Yaskawa INFORM job: s1234_1.JBI

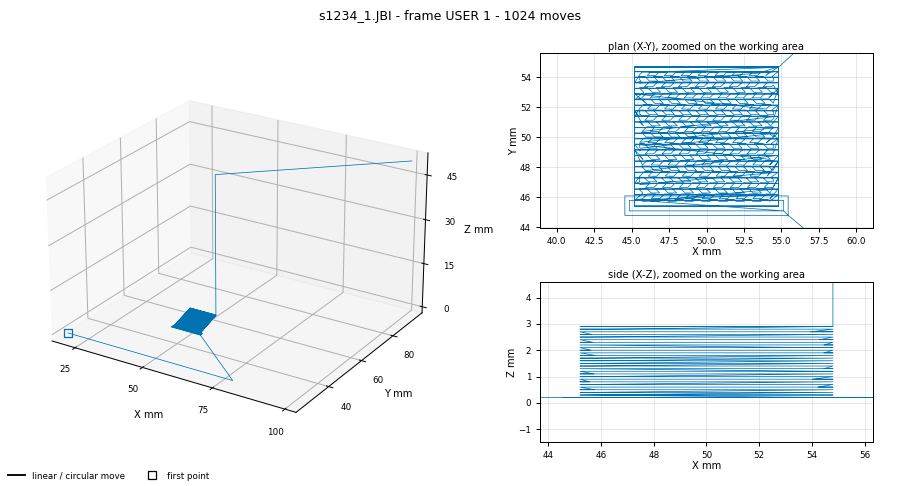
[picture p0: tool path of s1234_1.JBI in frame USER 1, 1024 of 1024 moves have a stored position in this frame; points joined in program order, loops and branches not executed]
/JOB
//NAME s1234_1
//POS
///NPOS 1024,0,0,0,0,0
///USER 1
///TOOL 1
///POSTYPE USER
///RECTAN
///RCONF 1,0,0,0,0,0
C00000=20.000,24.400,0.200,0.000,-180.000,-30.000
C00001=80.000,24.400,0.200,0.000,-180.000,-30.000
C00002=80.000,24.400,0.200,0.000,-180.000,-30.000
C00003=55.450,44.784,0.200,0.000,-180.000,-30.000
C00004=55.450,44.784,0.200,0.000,-180.000,-30.000
C00005=55.450,46.080,0.200,0.000,-180.000,-30.000
C00006=44.550,46.080,0.200,0.000,-180.000,-30.000
C00007=44.550,44.784,0.200,0.000,-180.000,-30.000
C00008=55.450,44.784,0.200,0.000,-180.000,-30.000
C00009=55.150,45.084,0.200,0.000,-180.000,-30.000
C00010=55.150,45.780,0.200,0.000,-180.000,-30.000
C00011=44.850,45.780,0.200,0.000,-180.000,-30.000
C00012=44.850,45.084,0.200,0.000,-180.000,-30.000
C00013=55.150,45.084,0.200,0.000,-180.000,-30.000
C00014=55.150,45.084,0.200,0.000,-180.000,-30.000
C00015=45.200,45.803,0.300,0.000,-180.000,-30.000
C00016=45.200,45.803,0.300,0.000,-180.000,-30.000
C00017=45.200,45.407,0.300,0.000,-180.000,-30.000
C00018=54.800,45.407,0.300,0.000,-180.000,-30.000
C00019=54.800,45.803,0.300,0.000,-180.000,-30.000
C00020=45.200,45.803,0.300,0.000,-180.000,-30.000
C00021=45.200,45.803,0.300,0.000,-180.000,-30.000
C00022=54.800,46.176,0.400,0.000,-180.000,-30.000
C00023=54.800,46.176,0.400,0.000,-180.000,-30.000
C00024=45.200,46.176,0.400,0.000,-180.000,-30.000
C00025=45.200,45.380,0.400,0.000,-180.000,-30.000
C00026=54.800,45.380,0.400,0.000,-180.000,-30.000
C00027=54.800,46.176,0.400,0.000,-180.000,-30.000
C00028=54.221,45.720,0.400,0.000,-180.000,-30.000
C00029=54.105,45.836,0.400,0.000,-180.000,-30.000
C00030=53.539,45.836,0.400,0.000,-180.000,-30.000
C00031=53.655,45.720,0.400,0.000,-180.000,-30.000
C00032=53.090,45.720,0.400,0.000,-180.000,-30.000
C00033=52.974,45.836,0.400,0.000,-180.000,-30.000
C00034=52.408,45.836,0.400,0.000,-180.000,-30.000
C00035=52.524,45.720,0.400,0.000,-180.000,-30.000
C00036=51.958,45.720,0.400,0.000,-180.000,-30.000
C00037=51.842,45.836,0.400,0.000,-180.000,-30.000
C00038=51.277,45.836,0.400,0.000,-180.000,-30.000
C00039=51.393,45.720,0.400,0.000,-180.000,-30.000
C00040=50.827,45.720,0.400,0.000,-180.000,-30.000
C00041=50.711,45.836,0.400,0.000,-180.000,-30.000
C00042=50.145,45.836,0.400,0.000,-180.000,-30.000
C00043=50.261,45.720,0.400,0.000,-180.000,-30.000
C00044=49.696,45.720,0.400,0.000,-180.000,-30.000
C00045=49.580,45.836,0.400,0.000,-180.000,-30.000
C00046=49.014,45.836,0.400,0.000,-180.000,-30.000
C00047=49.130,45.720,0.400,0.000,-180.000,-30.000
C00048=48.564,45.720,0.400,0.000,-180.000,-30.000
C00049=48.448,45.836,0.400,0.000,-180.000,-30.000
C00050=47.883,45.836,0.400,0.000,-180.000,-30.000
C00051=47.999,45.720,0.400,0.000,-180.000,-30.000
C00052=47.433,45.720,0.400,0.000,-180.000,-30.000
C00053=47.317,45.836,0.400,0.000,-180.000,-30.000
C00054=46.751,45.836,0.400,0.000,-180.000,-30.000
C00055=46.867,45.720,0.400,0.000,-180.000,-30.000
C00056=46.302,45.720,0.400,0.000,-180.000,-30.000
C00057=46.186,45.836,0.400,0.000,-180.000,-30.000
C00058=45.620,45.836,0.400,0.000,-180.000,-30.000
C00059=45.736,45.720,0.400,0.000,-180.000,-30.000
C00060=45.736,45.720,0.400,0.000,-180.000,-30.000
C00061=54.800,46.550,0.500,0.000,-180.000,-30.000
C00062=54.800,46.550,0.500,0.000,-180.000,-30.000
C00063=45.200,46.550,0.500,0.000,-180.000,-30.000
C00064=45.200,45.409,0.500,0.000,-180.000,-30.000
C00065=54.800,45.409,0.500,0.000,-180.000,-30.000
C00066=54.800,46.550,0.500,0.000,-180.000,-30.000
C00067=54.800,46.550,0.500,0.000,-180.000,-30.000
C00068=54.232,45.903,0.500,0.000,-180.000,-30.000
C00069=54.232,45.903,0.500,0.000,-180.000,-30.000
C00070=54.460,46.131,0.500,0.000,-180.000,-30.000
C00071=54.460,46.210,0.500,0.000,-180.000,-30.000
C00072=53.974,46.210,0.500,0.000,-180.000,-30.000
C00073=53.667,45.903,0.500,0.000,-180.000,-30.000
C00074=53.101,45.903,0.500,0.000,-180.000,-30.000
C00075=53.408,46.210,0.500,0.000,-180.000,-30.000
C00076=52.842,46.210,0.500,0.000,-180.000,-30.000
C00077=52.535,45.903,0.500,0.000,-180.000,-30.000
C00078=51.970,45.903,0.500,0.000,-180.000,-30.000
C00079=52.277,46.210,0.500,0.000,-180.000,-30.000
C00080=51.711,46.210,0.500,0.000,-180.000,-30.000
C00081=51.404,45.903,0.500,0.000,-180.000,-30.000
C00082=50.838,45.903,0.500,0.000,-180.000,-30.000
C00083=51.145,46.210,0.500,0.000,-180.000,-30.000
C00084=50.580,46.210,0.500,0.000,-180.000,-30.000
C00085=50.273,45.903,0.500,0.000,-180.000,-30.000
C00086=49.707,45.903,0.500,0.000,-180.000,-30.000
C00087=50.014,46.210,0.500,0.000,-180.000,-30.000
C00088=49.448,46.210,0.500,0.000,-180.000,-30.000
C00089=49.141,45.903,0.500,0.000,-180.000,-30.000
C00090=48.576,45.903,0.500,0.000,-180.000,-30.000
C00091=48.883,46.210,0.500,0.000,-180.000,-30.000
C00092=48.317,46.210,0.500,0.000,-180.000,-30.000
C00093=48.010,45.903,0.500,0.000,-180.000,-30.000
C00094=47.444,45.903,0.500,0.000,-180.000,-30.000
C00095=47.751,46.210,0.500,0.000,-180.000,-30.000
C00096=47.186,46.210,0.500,0.000,-180.000,-30.000
C00097=46.879,45.903,0.500,0.000,-180.000,-30.000
C00098=46.313,45.903,0.500,0.000,-180.000,-30.000
C00099=46.620,46.210,0.500,0.000,-180.000,-30.000
C00100=46.054,46.210,0.500,0.000,-180.000,-30.000
C00101=45.747,45.903,0.500,0.000,-180.000,-30.000
C00102=45.747,45.903,0.500,0.000,-180.000,-30.000
C00103=45.200,45.782,0.600,0.000,-180.000,-30.000
C00104=45.200,45.782,0.600,0.000,-180.000,-30.000
C00105=54.800,45.782,0.600,0.000,-180.000,-30.000
C00106=54.800,46.923,0.600,0.000,-180.000,-30.000
C00107=45.200,46.923,0.600,0.000,-180.000,-30.000
C00108=45.200,45.782,0.600,0.000,-180.000,-30.000
C00109=45.746,46.276,0.600,0.000,-180.000,-30.000
C00110=45.540,46.482,0.600,0.000,-180.000,-30.000
C00111=45.540,46.583,0.600,0.000,-180.000,-30.000
C00112=46.004,46.583,0.600,0.000,-180.000,-30.000
C00113=46.311,46.276,0.600,0.000,-180.000,-30.000
C00114=46.877,46.276,0.600,0.000,-180.000,-30.000
C00115=46.570,46.583,0.600,0.000,-180.000,-30.000
C00116=47.136,46.583,0.600,0.000,-180.000,-30.000
C00117=47.443,46.276,0.600,0.000,-180.000,-30.000
C00118=48.008,46.276,0.600,0.000,-180.000,-30.000
C00119=47.701,46.583,0.600,0.000,-180.000,-30.000
C00120=48.267,46.583,0.600,0.000,-180.000,-30.000
C00121=48.574,46.276,0.600,0.000,-180.000,-30.000
C00122=49.140,46.276,0.600,0.000,-180.000,-30.000
C00123=48.833,46.583,0.600,0.000,-180.000,-30.000
C00124=49.398,46.583,0.600,0.000,-180.000,-30.000
C00125=49.705,46.276,0.600,0.000,-180.000,-30.000
C00126=50.271,46.276,0.600,0.000,-180.000,-30.000
C00127=49.964,46.583,0.600,0.000,-180.000,-30.000
C00128=50.530,46.583,0.600,0.000,-180.000,-30.000
C00129=50.837,46.276,0.600,0.000,-180.000,-30.000
C00130=51.402,46.276,0.600,0.000,-180.000,-30.000
C00131=51.095,46.583,0.600,0.000,-180.000,-30.000
C00132=51.661,46.583,0.600,0.000,-180.000,-30.000
C00133=51.968,46.276,0.600,0.000,-180.000,-30.000
C00134=52.534,46.276,0.600,0.000,-180.000,-30.000
C00135=52.227,46.583,0.600,0.000,-180.000,-30.000
C00136=52.792,46.583,0.600,0.000,-180.000,-30.000
C00137=53.099,46.276,0.600,0.000,-180.000,-30.000
C00138=53.665,46.276,0.600,0.000,-180.000,-30.000
C00139=53.358,46.583,0.600,0.000,-180.000,-30.000
C00140=53.924,46.583,0.600,0.000,-180.000,-30.000
C00141=54.231,46.276,0.600,0.000,-180.000,-30.000
C00142=54.231,46.276,0.600,0.000,-180.000,-30.000
C00143=54.800,47.297,0.700,0.000,-180.000,-30.000
C00144=54.800,47.297,0.700,0.000,-180.000,-30.000
C00145=45.200,47.297,0.700,0.000,-180.000,-30.000
C00146=45.200,46.155,0.700,0.000,-180.000,-30.000
C00147=54.800,46.155,0.700,0.000,-180.000,-30.000
C00148=54.800,47.297,0.700,0.000,-180.000,-30.000
C00149=54.460,46.696,0.700,0.000,-180.000,-30.000
C00150=54.414,46.650,0.700,0.000,-180.000,-30.000
C00151=53.848,46.650,0.700,0.000,-180.000,-30.000
C00152=54.155,46.957,0.700,0.000,-180.000,-30.000
C00153=53.589,46.957,0.700,0.000,-180.000,-30.000
C00154=53.282,46.650,0.700,0.000,-180.000,-30.000
C00155=52.717,46.650,0.700,0.000,-180.000,-30.000
C00156=53.024,46.957,0.700,0.000,-180.000,-30.000
C00157=52.458,46.957,0.700,0.000,-180.000,-30.000
C00158=52.151,46.650,0.700,0.000,-180.000,-30.000
C00159=51.585,46.650,0.700,0.000,-180.000,-30.000
C00160=51.892,46.957,0.700,0.000,-180.000,-30.000
C00161=51.327,46.957,0.700,0.000,-180.000,-30.000
C00162=51.020,46.650,0.700,0.000,-180.000,-30.000
C00163=50.454,46.650,0.700,0.000,-180.000,-30.000
C00164=50.761,46.957,0.700,0.000,-180.000,-30.000
C00165=50.195,46.957,0.700,0.000,-180.000,-30.000
C00166=49.888,46.650,0.700,0.000,-180.000,-30.000
C00167=49.323,46.650,0.700,0.000,-180.000,-30.000
C00168=49.630,46.957,0.700,0.000,-180.000,-30.000
C00169=49.064,46.957,0.700,0.000,-180.000,-30.000
C00170=48.757,46.650,0.700,0.000,-180.000,-30.000
C00171=48.191,46.650,0.700,0.000,-180.000,-30.000
C00172=48.498,46.957,0.700,0.000,-180.000,-30.000
C00173=47.933,46.957,0.700,0.000,-180.000,-30.000
C00174=47.626,46.650,0.700,0.000,-180.000,-30.000
C00175=47.060,46.650,0.700,0.000,-180.000,-30.000
C00176=47.367,46.957,0.700,0.000,-180.000,-30.000
C00177=46.801,46.957,0.700,0.000,-180.000,-30.000
C00178=46.494,46.650,0.700,0.000,-180.000,-30.000
C00179=45.928,46.650,0.700,0.000,-180.000,-30.000
C00180=46.235,46.957,0.700,0.000,-180.000,-30.000
C00181=45.670,46.957,0.700,0.000,-180.000,-30.000
C00182=45.540,46.827,0.700,0.000,-180.000,-30.000
C00183=45.540,46.827,0.700,0.000,-180.000,-30.000
C00184=54.800,47.670,0.800,0.000,-180.000,-30.000
C00185=54.800,47.670,0.800,0.000,-180.000,-30.000
C00186=45.200,47.670,0.800,0.000,-180.000,-30.000
C00187=45.200,46.528,0.800,0.000,-180.000,-30.000
C00188=54.800,46.528,0.800,0.000,-180.000,-30.000
C00189=54.800,47.670,0.800,0.000,-180.000,-30.000
C00190=54.308,47.330,0.800,0.000,-180.000,-30.000
C00191=54.460,47.178,0.800,0.000,-180.000,-30.000
C00192=54.460,47.023,0.800,0.000,-180.000,-30.000
C00193=54.050,47.023,0.800,0.000,-180.000,-30.000
C00194=53.743,47.330,0.800,0.000,-180.000,-30.000
C00195=53.177,47.330,0.800,0.000,-180.000,-30.000
C00196=53.484,47.023,0.800,0.000,-180.000,-30.000
C00197=52.918,47.023,0.800,0.000,-180.000,-30.000
C00198=52.611,47.330,0.800,0.000,-180.000,-30.000
C00199=52.045,47.330,0.800,0.000,-180.000,-30.000
C00200=52.352,47.023,0.800,0.000,-180.000,-30.000
C00201=51.787,47.023,0.800,0.000,-180.000,-30.000
C00202=51.480,47.330,0.800,0.000,-180.000,-30.000
C00203=50.914,47.330,0.800,0.000,-180.000,-30.000
C00204=51.221,47.023,0.800,0.000,-180.000,-30.000
C00205=50.655,47.023,0.800,0.000,-180.000,-30.000
C00206=50.348,47.330,0.800,0.000,-180.000,-30.000
C00207=49.783,47.330,0.800,0.000,-180.000,-30.000
C00208=50.090,47.023,0.800,0.000,-180.000,-30.000
C00209=49.524,47.023,0.800,0.000,-180.000,-30.000
C00210=49.217,47.330,0.800,0.000,-180.000,-30.000
C00211=48.651,47.330,0.800,0.000,-180.000,-30.000
C00212=48.958,47.023,0.800,0.000,-180.000,-30.000
C00213=48.393,47.023,0.800,0.000,-180.000,-30.000
C00214=48.086,47.330,0.800,0.000,-180.000,-30.000
C00215=47.520,47.330,0.800,0.000,-180.000,-30.000
C00216=47.827,47.023,0.800,0.000,-180.000,-30.000
C00217=47.261,47.023,0.800,0.000,-180.000,-30.000
C00218=46.954,47.330,0.800,0.000,-180.000,-30.000
C00219=46.389,47.330,0.800,0.000,-180.000,-30.000
C00220=46.696,47.023,0.800,0.000,-180.000,-30.000
C00221=46.130,47.023,0.800,0.000,-180.000,-30.000
C00222=45.823,47.330,0.800,0.000,-180.000,-30.000
C00223=45.540,47.330,0.800,0.000,-180.000,-30.000
C00224=45.540,47.047,0.800,0.000,-180.000,-30.000
C00225=45.564,47.023,0.800,0.000,-180.000,-30.000
C00226=45.564,47.023,0.800,0.000,-180.000,-30.000
C00227=45.200,46.902,0.900,0.000,-180.000,-30.000
C00228=45.200,46.902,0.900,0.000,-180.000,-30.000
C00229=54.800,46.902,0.900,0.000,-180.000,-30.000
C00230=54.800,48.044,0.900,0.000,-180.000,-30.000
C00231=45.200,48.044,0.900,0.000,-180.000,-30.000
C00232=45.200,46.902,0.900,0.000,-180.000,-30.000
C00233=45.544,47.397,0.900,0.000,-180.000,-30.000
C00234=45.851,47.704,0.900,0.000,-180.000,-30.000
C00235=46.417,47.704,0.900,0.000,-180.000,-30.000
C00236=46.110,47.397,0.900,0.000,-180.000,-30.000
C00237=46.675,47.397,0.900,0.000,-180.000,-30.000
C00238=46.982,47.704,0.900,0.000,-180.000,-30.000
C00239=47.548,47.704,0.900,0.000,-180.000,-30.000
C00240=47.241,47.397,0.900,0.000,-180.000,-30.000
C00241=47.807,47.397,0.900,0.000,-180.000,-30.000
C00242=48.114,47.704,0.900,0.000,-180.000,-30.000
C00243=48.680,47.704,0.900,0.000,-180.000,-30.000
C00244=48.373,47.397,0.900,0.000,-180.000,-30.000
C00245=48.938,47.397,0.900,0.000,-180.000,-30.000
C00246=49.245,47.704,0.900,0.000,-180.000,-30.000
C00247=49.811,47.704,0.900,0.000,-180.000,-30.000
C00248=49.504,47.397,0.900,0.000,-180.000,-30.000
C00249=50.070,47.397,0.900,0.000,-180.000,-30.000
C00250=50.377,47.704,0.900,0.000,-180.000,-30.000
C00251=50.942,47.704,0.900,0.000,-180.000,-30.000
C00252=50.635,47.397,0.900,0.000,-180.000,-30.000
C00253=51.201,47.397,0.900,0.000,-180.000,-30.000
C00254=51.508,47.704,0.900,0.000,-180.000,-30.000
C00255=52.074,47.704,0.900,0.000,-180.000,-30.000
C00256=51.767,47.397,0.900,0.000,-180.000,-30.000
C00257=52.332,47.397,0.900,0.000,-180.000,-30.000
C00258=52.639,47.704,0.900,0.000,-180.000,-30.000
C00259=53.205,47.704,0.900,0.000,-180.000,-30.000
C00260=52.898,47.397,0.900,0.000,-180.000,-30.000
C00261=53.464,47.397,0.900,0.000,-180.000,-30.000
C00262=53.771,47.704,0.900,0.000,-180.000,-30.000
C00263=54.336,47.704,0.900,0.000,-180.000,-30.000
C00264=54.029,47.397,0.900,0.000,-180.000,-30.000
C00265=54.029,47.397,0.900,0.000,-180.000,-30.000
C00266=54.800,48.417,1.000,0.000,-180.000,-30.000
C00267=54.800,48.417,1.000,0.000,-180.000,-30.000
C00268=45.200,48.417,1.000,0.000,-180.000,-30.000
C00269=45.200,47.275,1.000,0.000,-180.000,-30.000
C00270=54.800,47.275,1.000,0.000,-180.000,-30.000
C00271=54.800,48.417,1.000,0.000,-180.000,-30.000
C00272=54.434,47.770,1.000,0.000,-180.000,-30.000
C00273=54.127,48.077,1.000,0.000,-180.000,-30.000
C00274=53.561,48.077,1.000,0.000,-180.000,-30.000
C00275=53.868,47.770,1.000,0.000,-180.000,-30.000
C00276=53.303,47.770,1.000,0.000,-180.000,-30.000
C00277=52.996,48.077,1.000,0.000,-180.000,-30.000
C00278=52.430,48.077,1.000,0.000,-180.000,-30.000
C00279=52.737,47.770,1.000,0.000,-180.000,-30.000
C00280=52.171,47.770,1.000,0.000,-180.000,-30.000
C00281=51.864,48.077,1.000,0.000,-180.000,-30.000
C00282=51.298,48.077,1.000,0.000,-180.000,-30.000
C00283=51.605,47.770,1.000,0.000,-180.000,-30.000
C00284=51.040,47.770,1.000,0.000,-180.000,-30.000
C00285=50.733,48.077,1.000,0.000,-180.000,-30.000
C00286=50.167,48.077,1.000,0.000,-180.000,-30.000
C00287=50.474,47.770,1.000,0.000,-180.000,-30.000
C00288=49.908,47.770,1.000,0.000,-180.000,-30.000
C00289=49.601,48.077,1.000,0.000,-180.000,-30.000
C00290=49.036,48.077,1.000,0.000,-180.000,-30.000
C00291=49.343,47.770,1.000,0.000,-180.000,-30.000
C00292=48.777,47.770,1.000,0.000,-180.000,-30.000
C00293=48.470,48.077,1.000,0.000,-180.000,-30.000
C00294=47.904,48.077,1.000,0.000,-180.000,-30.000
C00295=48.211,47.770,1.000,0.000,-180.000,-30.000
C00296=47.646,47.770,1.000,0.000,-180.000,-30.000
C00297=47.339,48.077,1.000,0.000,-180.000,-30.000
C00298=46.773,48.077,1.000,0.000,-180.000,-30.000
C00299=47.080,47.770,1.000,0.000,-180.000,-30.000
C00300=46.514,47.770,1.000,0.000,-180.000,-30.000
C00301=46.207,48.077,1.000,0.000,-180.000,-30.000
C00302=45.642,48.077,1.000,0.000,-180.000,-30.000
C00303=45.949,47.770,1.000,0.000,-180.000,-30.000
C00304=45.949,47.770,1.000,0.000,-180.000,-30.000
C00305=54.800,48.790,1.100,0.000,-180.000,-30.000
C00306=54.800,48.790,1.100,0.000,-180.000,-30.000
C00307=45.200,48.790,1.100,0.000,-180.000,-30.000
C00308=45.200,47.648,1.100,0.000,-180.000,-30.000
C00309=54.800,47.648,1.100,0.000,-180.000,-30.000
C00310=54.800,48.790,1.100,0.000,-180.000,-30.000
C00311=54.800,48.790,1.100,0.000,-180.000,-30.000
C00312=54.211,48.144,1.100,0.000,-180.000,-30.000
C00313=54.211,48.144,1.100,0.000,-180.000,-30.000
C00314=54.460,48.393,1.100,0.000,-180.000,-30.000
C00315=54.460,48.450,1.100,0.000,-180.000,-30.000
C00316=53.951,48.450,1.100,0.000,-180.000,-30.000
C00317=53.645,48.144,1.100,0.000,-180.000,-30.000
C00318=53.079,48.144,1.100,0.000,-180.000,-30.000
C00319=53.385,48.450,1.100,0.000,-180.000,-30.000
C00320=52.820,48.450,1.100,0.000,-180.000,-30.000
C00321=52.514,48.144,1.100,0.000,-180.000,-30.000
C00322=51.948,48.144,1.100,0.000,-180.000,-30.000
C00323=52.254,48.450,1.100,0.000,-180.000,-30.000
C00324=51.688,48.450,1.100,0.000,-180.000,-30.000
C00325=51.382,48.144,1.100,0.000,-180.000,-30.000
C00326=50.817,48.144,1.100,0.000,-180.000,-30.000
C00327=51.123,48.450,1.100,0.000,-180.000,-30.000
C00328=50.557,48.450,1.100,0.000,-180.000,-30.000
C00329=50.251,48.144,1.100,0.000,-180.000,-30.000
C00330=49.685,48.144,1.100,0.000,-180.000,-30.000
C00331=49.991,48.450,1.100,0.000,-180.000,-30.000
C00332=49.426,48.450,1.100,0.000,-180.000,-30.000
C00333=49.120,48.144,1.100,0.000,-180.000,-30.000
C00334=48.554,48.144,1.100,0.000,-180.000,-30.000
C00335=48.860,48.450,1.100,0.000,-180.000,-30.000
C00336=48.294,48.450,1.100,0.000,-180.000,-30.000
C00337=47.988,48.144,1.100,0.000,-180.000,-30.000
C00338=47.422,48.144,1.100,0.000,-180.000,-30.000
C00339=47.728,48.450,1.100,0.000,-180.000,-30.000
C00340=47.163,48.450,1.100,0.000,-180.000,-30.000
C00341=46.857,48.144,1.100,0.000,-180.000,-30.000
C00342=46.291,48.144,1.100,0.000,-180.000,-30.000
C00343=46.597,48.450,1.100,0.000,-180.000,-30.000
C00344=46.031,48.450,1.100,0.000,-180.000,-30.000
C00345=45.725,48.144,1.100,0.000,-180.000,-30.000
C00346=45.725,48.144,1.100,0.000,-180.000,-30.000
C00347=45.200,49.164,1.200,0.000,-180.000,-30.000
C00348=45.200,49.164,1.200,0.000,-180.000,-30.000
C00349=45.200,48.021,1.200,0.000,-180.000,-30.000
C00350=54.800,48.021,1.200,0.000,-180.000,-30.000
C00351=54.800,49.164,1.200,0.000,-180.000,-30.000
C00352=45.200,49.164,1.200,0.000,-180.000,-30.000
C00353=45.200,49.164,1.200,0.000,-180.000,-30.000
C00354=45.767,48.517,1.200,0.000,-180.000,-30.000
C00355=45.767,48.517,1.200,0.000,-180.000,-30.000
C00356=45.540,48.744,1.200,0.000,-180.000,-30.000
C00357=45.540,48.824,1.200,0.000,-180.000,-30.000
C00358=46.026,48.824,1.200,0.000,-180.000,-30.000
C00359=46.333,48.517,1.200,0.000,-180.000,-30.000
C00360=46.899,48.517,1.200,0.000,-180.000,-30.000
C00361=46.592,48.824,1.200,0.000,-180.000,-30.000
C00362=47.157,48.824,1.200,0.000,-180.000,-30.000
C00363=47.464,48.517,1.200,0.000,-180.000,-30.000
C00364=48.030,48.517,1.200,0.000,-180.000,-30.000
C00365=47.723,48.824,1.200,0.000,-180.000,-30.000
C00366=48.289,48.824,1.200,0.000,-180.000,-30.000
C00367=48.596,48.517,1.200,0.000,-180.000,-30.000
C00368=49.161,48.517,1.200,0.000,-180.000,-30.000
C00369=48.854,48.824,1.200,0.000,-180.000,-30.000
C00370=49.420,48.824,1.200,0.000,-180.000,-30.000
C00371=49.727,48.517,1.200,0.000,-180.000,-30.000
C00372=50.293,48.517,1.200,0.000,-180.000,-30.000
C00373=49.986,48.824,1.200,0.000,-180.000,-30.000
C00374=50.551,48.824,1.200,0.000,-180.000,-30.000
C00375=50.858,48.517,1.200,0.000,-180.000,-30.000
C00376=51.424,48.517,1.200,0.000,-180.000,-30.000
C00377=51.117,48.824,1.200,0.000,-180.000,-30.000
C00378=51.683,48.824,1.200,0.000,-180.000,-30.000
C00379=51.990,48.517,1.200,0.000,-180.000,-30.000
C00380=52.556,48.517,1.200,0.000,-180.000,-30.000
C00381=52.249,48.824,1.200,0.000,-180.000,-30.000
C00382=52.814,48.824,1.200,0.000,-180.000,-30.000
C00383=53.121,48.517,1.200,0.000,-180.000,-30.000
C00384=53.687,48.517,1.200,0.000,-180.000,-30.000
C00385=53.380,48.824,1.200,0.000,-180.000,-30.000
C00386=53.946,48.824,1.200,0.000,-180.000,-30.000
C00387=54.253,48.517,1.200,0.000,-180.000,-30.000
C00388=54.253,48.517,1.200,0.000,-180.000,-30.000
C00389=45.200,49.537,1.300,0.000,-180.000,-30.000
C00390=45.200,49.537,1.300,0.000,-180.000,-30.000
C00391=45.200,48.394,1.300,0.000,-180.000,-30.000
C00392=54.800,48.394,1.300,0.000,-180.000,-30.000
C00393=54.800,49.537,1.300,0.000,-180.000,-30.000
C00394=45.200,49.537,1.300,0.000,-180.000,-30.000
C00395=45.540,49.090,1.300,0.000,-180.000,-30.000
C00396=45.647,49.197,1.300,0.000,-180.000,-30.000
C00397=46.213,49.197,1.300,0.000,-180.000,-30.000
C00398=45.906,48.890,1.300,0.000,-180.000,-30.000
C00399=46.471,48.890,1.300,0.000,-180.000,-30.000
C00400=46.778,49.197,1.300,0.000,-180.000,-30.000
C00401=47.344,49.197,1.300,0.000,-180.000,-30.000
C00402=47.037,48.890,1.300,0.000,-180.000,-30.000
C00403=47.603,48.890,1.300,0.000,-180.000,-30.000
C00404=47.910,49.197,1.300,0.000,-180.000,-30.000
C00405=48.475,49.197,1.300,0.000,-180.000,-30.000
C00406=48.168,48.890,1.300,0.000,-180.000,-30.000
C00407=48.734,48.890,1.300,0.000,-180.000,-30.000
C00408=49.041,49.197,1.300,0.000,-180.000,-30.000
C00409=49.607,49.197,1.300,0.000,-180.000,-30.000
C00410=49.300,48.890,1.300,0.000,-180.000,-30.000
C00411=49.866,48.890,1.300,0.000,-180.000,-30.000
C00412=50.173,49.197,1.300,0.000,-180.000,-30.000
C00413=50.738,49.197,1.300,0.000,-180.000,-30.000
C00414=50.431,48.890,1.300,0.000,-180.000,-30.000
C00415=50.997,48.890,1.300,0.000,-180.000,-30.000
C00416=51.304,49.197,1.300,0.000,-180.000,-30.000
C00417=51.870,49.197,1.300,0.000,-180.000,-30.000
C00418=51.563,48.890,1.300,0.000,-180.000,-30.000
C00419=52.128,48.890,1.300,0.000,-180.000,-30.000
C00420=52.435,49.197,1.300,0.000,-180.000,-30.000
C00421=53.001,49.197,1.300,0.000,-180.000,-30.000
C00422=52.694,48.890,1.300,0.000,-180.000,-30.000
C00423=53.260,48.890,1.300,0.000,-180.000,-30.000
C00424=53.567,49.197,1.300,0.000,-180.000,-30.000
C00425=54.132,49.197,1.300,0.000,-180.000,-30.000
C00426=53.825,48.890,1.300,0.000,-180.000,-30.000
C00427=54.391,48.890,1.300,0.000,-180.000,-30.000
C00428=54.460,48.959,1.300,0.000,-180.000,-30.000
C00429=54.460,48.959,1.300,0.000,-180.000,-30.000
C00430=54.800,49.911,1.400,0.000,-180.000,-30.000
C00431=54.800,49.911,1.400,0.000,-180.000,-30.000
C00432=45.200,49.911,1.400,0.000,-180.000,-30.000
C00433=45.200,48.767,1.400,0.000,-180.000,-30.000
C00434=54.800,48.767,1.400,0.000,-180.000,-30.000
C00435=54.800,49.911,1.400,0.000,-180.000,-30.000
C00436=54.330,49.571,1.400,0.000,-180.000,-30.000
C00437=54.460,49.441,1.400,0.000,-180.000,-30.000
C00438=54.460,49.264,1.400,0.000,-180.000,-30.000
C00439=54.071,49.264,1.400,0.000,-180.000,-30.000
C00440=53.764,49.571,1.400,0.000,-180.000,-30.000
C00441=53.199,49.571,1.400,0.000,-180.000,-30.000
C00442=53.506,49.264,1.400,0.000,-180.000,-30.000
C00443=52.940,49.264,1.400,0.000,-180.000,-30.000
C00444=52.633,49.571,1.400,0.000,-180.000,-30.000
C00445=52.067,49.571,1.400,0.000,-180.000,-30.000
C00446=52.374,49.264,1.400,0.000,-180.000,-30.000
C00447=51.809,49.264,1.400,0.000,-180.000,-30.000
C00448=51.502,49.571,1.400,0.000,-180.000,-30.000
C00449=50.936,49.571,1.400,0.000,-180.000,-30.000
C00450=51.243,49.264,1.400,0.000,-180.000,-30.000
C00451=50.677,49.264,1.400,0.000,-180.000,-30.000
C00452=50.370,49.571,1.400,0.000,-180.000,-30.000
C00453=49.804,49.571,1.400,0.000,-180.000,-30.000
C00454=50.111,49.264,1.400,0.000,-180.000,-30.000
C00455=49.546,49.264,1.400,0.000,-180.000,-30.000
C00456=49.239,49.571,1.400,0.000,-180.000,-30.000
C00457=48.673,49.571,1.400,0.000,-180.000,-30.000
C00458=48.980,49.264,1.400,0.000,-180.000,-30.000
C00459=48.414,49.264,1.400,0.000,-180.000,-30.000
C00460=48.107,49.571,1.400,0.000,-180.000,-30.000
C00461=47.542,49.571,1.400,0.000,-180.000,-30.000
C00462=47.849,49.264,1.400,0.000,-180.000,-30.000
C00463=47.283,49.264,1.400,0.000,-180.000,-30.000
C00464=46.976,49.571,1.400,0.000,-180.000,-30.000
C00465=46.410,49.571,1.400,0.000,-180.000,-30.000
C00466=46.717,49.264,1.400,0.000,-180.000,-30.000
C00467=46.152,49.264,1.400,0.000,-180.000,-30.000
C00468=45.845,49.571,1.400,0.000,-180.000,-30.000
C00469=45.540,49.571,1.400,0.000,-180.000,-30.000
C00470=45.540,49.310,1.400,0.000,-180.000,-30.000
C00471=45.586,49.264,1.400,0.000,-180.000,-30.000
C00472=45.586,49.264,1.400,0.000,-180.000,-30.000
C00473=54.800,50.284,1.500,0.000,-180.000,-30.000
C00474=54.800,50.284,1.500,0.000,-180.000,-30.000
C00475=45.200,50.284,1.500,0.000,-180.000,-30.000
C00476=45.200,49.140,1.500,0.000,-180.000,-30.000
C00477=54.800,49.140,1.500,0.000,-180.000,-30.000
C00478=54.800,50.284,1.500,0.000,-180.000,-30.000
C00479=54.007,49.637,1.500,0.000,-180.000,-30.000
C00480=54.314,49.944,1.500,0.000,-180.000,-30.000
C00481=53.748,49.944,1.500,0.000,-180.000,-30.000
C00482=53.441,49.637,1.500,0.000,-180.000,-30.000
C00483=52.875,49.637,1.500,0.000,-180.000,-30.000
C00484=53.182,49.944,1.500,0.000,-180.000,-30.000
C00485=52.617,49.944,1.500,0.000,-180.000,-30.000
C00486=52.310,49.637,1.500,0.000,-180.000,-30.000
C00487=51.744,49.637,1.500,0.000,-180.000,-30.000
C00488=52.051,49.944,1.500,0.000,-180.000,-30.000
C00489=51.485,49.944,1.500,0.000,-180.000,-30.000
C00490=51.178,49.637,1.500,0.000,-180.000,-30.000
C00491=50.613,49.637,1.500,0.000,-180.000,-30.000
C00492=50.920,49.944,1.500,0.000,-180.000,-30.000
C00493=50.354,49.944,1.500,0.000,-180.000,-30.000
C00494=50.047,49.637,1.500,0.000,-180.000,-30.000
C00495=49.481,49.637,1.500,0.000,-180.000,-30.000
C00496=49.788,49.944,1.500,0.000,-180.000,-30.000
C00497=49.222,49.944,1.500,0.000,-180.000,-30.000
C00498=48.915,49.637,1.500,0.000,-180.000,-30.000
C00499=48.350,49.637,1.500,0.000,-180.000,-30.000
C00500=48.657,49.944,1.500,0.000,-180.000,-30.000
C00501=48.091,49.944,1.500,0.000,-180.000,-30.000
C00502=47.784,49.637,1.500,0.000,-180.000,-30.000
C00503=47.218,49.637,1.500,0.000,-180.000,-30.000
C00504=47.525,49.944,1.500,0.000,-180.000,-30.000
C00505=46.960,49.944,1.500,0.000,-180.000,-30.000
C00506=46.653,49.637,1.500,0.000,-180.000,-30.000
C00507=46.087,49.637,1.500,0.000,-180.000,-30.000
C00508=46.394,49.944,1.500,0.000,-180.000,-30.000
C00509=45.828,49.944,1.500,0.000,-180.000,-30.000
C00510=45.540,49.656,1.500,0.000,-180.000,-30.000
C00511=45.540,49.656,1.500,0.000,-180.000,-30.000
C00512=54.800,50.657,1.600,0.000,-180.000,-30.000
C00513=54.800,50.657,1.600,0.000,-180.000,-30.000
C00514=45.200,50.657,1.600,0.000,-180.000,-30.000
C00515=45.200,49.513,1.600,0.000,-180.000,-30.000
C00516=54.800,49.513,1.600,0.000,-180.000,-30.000
C00517=54.800,50.657,1.600,0.000,-180.000,-30.000
C00518=54.456,50.011,1.600,0.000,-180.000,-30.000
C00519=54.150,50.317,1.600,0.000,-180.000,-30.000
C00520=53.584,50.317,1.600,0.000,-180.000,-30.000
C00521=53.890,50.011,1.600,0.000,-180.000,-30.000
C00522=53.324,50.011,1.600,0.000,-180.000,-30.000
C00523=53.018,50.317,1.600,0.000,-180.000,-30.000
C00524=52.453,50.317,1.600,0.000,-180.000,-30.000
C00525=52.759,50.011,1.600,0.000,-180.000,-30.000
C00526=52.193,50.011,1.600,0.000,-180.000,-30.000
C00527=51.887,50.317,1.600,0.000,-180.000,-30.000
C00528=51.321,50.317,1.600,0.000,-180.000,-30.000
C00529=51.627,50.011,1.600,0.000,-180.000,-30.000
C00530=51.062,50.011,1.600,0.000,-180.000,-30.000
C00531=50.756,50.317,1.600,0.000,-180.000,-30.000
C00532=50.190,50.317,1.600,0.000,-180.000,-30.000
C00533=50.496,50.011,1.600,0.000,-180.000,-30.000
C00534=49.930,50.011,1.600,0.000,-180.000,-30.000
C00535=49.624,50.317,1.600,0.000,-180.000,-30.000
C00536=49.058,50.317,1.600,0.000,-180.000,-30.000
C00537=49.364,50.011,1.600,0.000,-180.000,-30.000
C00538=48.799,50.011,1.600,0.000,-180.000,-30.000
C00539=48.493,50.317,1.600,0.000,-180.000,-30.000
C00540=47.927,50.317,1.600,0.000,-180.000,-30.000
C00541=48.233,50.011,1.600,0.000,-180.000,-30.000
C00542=47.667,50.011,1.600,0.000,-180.000,-30.000
C00543=47.361,50.317,1.600,0.000,-180.000,-30.000
C00544=46.796,50.317,1.600,0.000,-180.000,-30.000
C00545=47.102,50.011,1.600,0.000,-180.000,-30.000
C00546=46.536,50.011,1.600,0.000,-180.000,-30.000
C00547=46.230,50.317,1.600,0.000,-180.000,-30.000
C00548=45.664,50.317,1.600,0.000,-180.000,-30.000
C00549=45.970,50.011,1.600,0.000,-180.000,-30.000
C00550=45.970,50.011,1.600,0.000,-180.000,-30.000
C00551=54.800,49.886,1.700,0.000,-180.000,-30.000
C00552=54.800,49.886,1.700,0.000,-180.000,-30.000
C00553=54.800,51.031,1.700,0.000,-180.000,-30.000
C00554=45.200,51.031,1.700,0.000,-180.000,-30.000
C00555=45.200,49.886,1.700,0.000,-180.000,-30.000
C00556=54.800,49.886,1.700,0.000,-180.000,-30.000
C00557=54.188,50.384,1.700,0.000,-180.000,-30.000
C00558=54.460,50.656,1.700,0.000,-180.000,-30.000
C00559=54.460,50.691,1.700,0.000,-180.000,-30.000
C00560=53.929,50.691,1.700,0.000,-180.000,-30.000
C00561=53.622,50.384,1.700,0.000,-180.000,-30.000
C00562=53.057,50.384,1.700,0.000,-180.000,-30.000
C00563=53.364,50.691,1.700,0.000,-180.000,-30.000
C00564=52.798,50.691,1.700,0.000,-180.000,-30.000
C00565=52.491,50.384,1.700,0.000,-180.000,-30.000
C00566=51.925,50.384,1.700,0.000,-180.000,-30.000
C00567=52.232,50.691,1.700,0.000,-180.000,-30.000
C00568=51.667,50.691,1.700,0.000,-180.000,-30.000
C00569=51.360,50.384,1.700,0.000,-180.000,-30.000
C00570=50.794,50.384,1.700,0.000,-180.000,-30.000
C00571=51.101,50.691,1.700,0.000,-180.000,-30.000
C00572=50.535,50.691,1.700,0.000,-180.000,-30.000
C00573=50.228,50.384,1.700,0.000,-180.000,-30.000
C00574=49.662,50.384,1.700,0.000,-180.000,-30.000
C00575=49.969,50.691,1.700,0.000,-180.000,-30.000
C00576=49.404,50.691,1.700,0.000,-180.000,-30.000
C00577=49.097,50.384,1.700,0.000,-180.000,-30.000
C00578=48.531,50.384,1.700,0.000,-180.000,-30.000
C00579=48.838,50.691,1.700,0.000,-180.000,-30.000
C00580=48.272,50.691,1.700,0.000,-180.000,-30.000
C00581=47.965,50.384,1.700,0.000,-180.000,-30.000
C00582=47.400,50.384,1.700,0.000,-180.000,-30.000
C00583=47.707,50.691,1.700,0.000,-180.000,-30.000
C00584=47.141,50.691,1.700,0.000,-180.000,-30.000
C00585=46.834,50.384,1.700,0.000,-180.000,-30.000
C00586=46.268,50.384,1.700,0.000,-180.000,-30.000
C00587=46.575,50.691,1.700,0.000,-180.000,-30.000
C00588=46.010,50.691,1.700,0.000,-180.000,-30.000
C00589=45.703,50.384,1.700,0.000,-180.000,-30.000
C00590=45.703,50.384,1.700,0.000,-180.000,-30.000
C00591=54.800,51.404,1.800,0.000,-180.000,-30.000
C00592=54.800,51.404,1.800,0.000,-180.000,-30.000
C00593=45.200,51.404,1.800,0.000,-180.000,-30.000
C00594=45.200,50.259,1.800,0.000,-180.000,-30.000
C00595=54.800,50.259,1.800,0.000,-180.000,-30.000
C00596=54.800,51.404,1.800,0.000,-180.000,-30.000
C00597=54.275,50.757,1.800,0.000,-180.000,-30.000
C00598=53.968,51.064,1.800,0.000,-180.000,-30.000
C00599=53.403,51.064,1.800,0.000,-180.000,-30.000
C00600=53.710,50.757,1.800,0.000,-180.000,-30.000
C00601=53.144,50.757,1.800,0.000,-180.000,-30.000
C00602=52.837,51.064,1.800,0.000,-180.000,-30.000
C00603=52.271,51.064,1.800,0.000,-180.000,-30.000
C00604=52.578,50.757,1.800,0.000,-180.000,-30.000
C00605=52.013,50.757,1.800,0.000,-180.000,-30.000
C00606=51.706,51.064,1.800,0.000,-180.000,-30.000
C00607=51.140,51.064,1.800,0.000,-180.000,-30.000
C00608=51.447,50.757,1.800,0.000,-180.000,-30.000
C00609=50.881,50.757,1.800,0.000,-180.000,-30.000
C00610=50.574,51.064,1.800,0.000,-180.000,-30.000
C00611=50.009,51.064,1.800,0.000,-180.000,-30.000
C00612=50.316,50.757,1.800,0.000,-180.000,-30.000
C00613=49.750,50.757,1.800,0.000,-180.000,-30.000
C00614=49.443,51.064,1.800,0.000,-180.000,-30.000
C00615=48.877,51.064,1.800,0.000,-180.000,-30.000
C00616=49.184,50.757,1.800,0.000,-180.000,-30.000
C00617=48.618,50.757,1.800,0.000,-180.000,-30.000
C00618=48.311,51.064,1.800,0.000,-180.000,-30.000
C00619=47.746,51.064,1.800,0.000,-180.000,-30.000
C00620=48.053,50.757,1.800,0.000,-180.000,-30.000
C00621=47.487,50.757,1.800,0.000,-180.000,-30.000
C00622=47.180,51.064,1.800,0.000,-180.000,-30.000
C00623=46.614,51.064,1.800,0.000,-180.000,-30.000
C00624=46.921,50.757,1.800,0.000,-180.000,-30.000
C00625=46.356,50.757,1.800,0.000,-180.000,-30.000
C00626=46.049,51.064,1.800,0.000,-180.000,-30.000
C00627=45.540,51.064,1.800,0.000,-180.000,-30.000
C00628=45.540,51.007,1.800,0.000,-180.000,-30.000
C00629=45.790,50.757,1.800,0.000,-180.000,-30.000
C00630=45.790,50.757,1.800,0.000,-180.000,-30.000
C00631=45.200,51.778,1.900,0.000,-180.000,-30.000
C00632=45.200,51.778,1.900,0.000,-180.000,-30.000
C00633=45.200,50.632,1.900,0.000,-180.000,-30.000
C00634=54.800,50.632,1.900,0.000,-180.000,-30.000
C00635=54.800,51.778,1.900,0.000,-180.000,-30.000
C00636=45.200,51.778,1.900,0.000,-180.000,-30.000
C00637=45.540,51.353,1.900,0.000,-180.000,-30.000
C00638=45.625,51.438,1.900,0.000,-180.000,-30.000
C00639=46.191,51.438,1.900,0.000,-180.000,-30.000
C00640=45.884,51.131,1.900,0.000,-180.000,-30.000
C00641=46.450,51.131,1.900,0.000,-180.000,-30.000
C00642=46.757,51.438,1.900,0.000,-180.000,-30.000
C00643=47.322,51.438,1.900,0.000,-180.000,-30.000
C00644=47.015,51.131,1.900,0.000,-180.000,-30.000
C00645=47.581,51.131,1.900,0.000,-180.000,-30.000
C00646=47.888,51.438,1.900,0.000,-180.000,-30.000
C00647=48.454,51.438,1.900,0.000,-180.000,-30.000
C00648=48.147,51.131,1.900,0.000,-180.000,-30.000
C00649=48.712,51.131,1.900,0.000,-180.000,-30.000
C00650=49.019,51.438,1.900,0.000,-180.000,-30.000
C00651=49.585,51.438,1.900,0.000,-180.000,-30.000
C00652=49.278,51.131,1.900,0.000,-180.000,-30.000
C00653=49.844,51.131,1.900,0.000,-180.000,-30.000
C00654=50.151,51.438,1.900,0.000,-180.000,-30.000
C00655=50.716,51.438,1.900,0.000,-180.000,-30.000
C00656=50.409,51.131,1.900,0.000,-180.000,-30.000
C00657=50.975,51.131,1.900,0.000,-180.000,-30.000
C00658=51.282,51.438,1.900,0.000,-180.000,-30.000
C00659=51.848,51.438,1.900,0.000,-180.000,-30.000
C00660=51.541,51.131,1.900,0.000,-180.000,-30.000
C00661=52.107,51.131,1.900,0.000,-180.000,-30.000
C00662=52.414,51.438,1.900,0.000,-180.000,-30.000
C00663=52.979,51.438,1.900,0.000,-180.000,-30.000
C00664=52.672,51.131,1.900,0.000,-180.000,-30.000
C00665=53.238,51.131,1.900,0.000,-180.000,-30.000
C00666=53.545,51.438,1.900,0.000,-180.000,-30.000
C00667=54.111,51.438,1.900,0.000,-180.000,-30.000
C00668=53.804,51.131,1.900,0.000,-180.000,-30.000
C00669=54.369,51.131,1.900,0.000,-180.000,-30.000
C00670=54.460,51.222,1.900,0.000,-180.000,-30.000
C00671=54.460,51.222,1.900,0.000,-180.000,-30.000
C00672=54.800,52.151,2.000,0.000,-180.000,-30.000
C00673=54.800,52.151,2.000,0.000,-180.000,-30.000
C00674=45.200,52.151,2.000,0.000,-180.000,-30.000
C00675=45.200,51.005,2.000,0.000,-180.000,-30.000
C00676=54.800,51.005,2.000,0.000,-180.000,-30.000
C00677=54.800,52.151,2.000,0.000,-180.000,-30.000
C00678=54.353,51.811,2.000,0.000,-180.000,-30.000
C00679=54.460,51.704,2.000,0.000,-180.000,-30.000
C00680=54.460,51.504,2.000,0.000,-180.000,-30.000
C00681=54.094,51.504,2.000,0.000,-180.000,-30.000
C00682=53.787,51.811,2.000,0.000,-180.000,-30.000
C00683=53.221,51.811,2.000,0.000,-180.000,-30.000
C00684=53.528,51.504,2.000,0.000,-180.000,-30.000
C00685=52.963,51.504,2.000,0.000,-180.000,-30.000
C00686=52.656,51.811,2.000,0.000,-180.000,-30.000
C00687=52.090,51.811,2.000,0.000,-180.000,-30.000
C00688=52.397,51.504,2.000,0.000,-180.000,-30.000
C00689=51.831,51.504,2.000,0.000,-180.000,-30.000
C00690=51.524,51.811,2.000,0.000,-180.000,-30.000
C00691=50.959,51.811,2.000,0.000,-180.000,-30.000
C00692=51.266,51.504,2.000,0.000,-180.000,-30.000
C00693=50.700,51.504,2.000,0.000,-180.000,-30.000
C00694=50.393,51.811,2.000,0.000,-180.000,-30.000
C00695=49.827,51.811,2.000,0.000,-180.000,-30.000
C00696=50.134,51.504,2.000,0.000,-180.000,-30.000
C00697=49.569,51.504,2.000,0.000,-180.000,-30.000
C00698=49.262,51.811,2.000,0.000,-180.000,-30.000
C00699=48.696,51.811,2.000,0.000,-180.000,-30.000
C00700=49.003,51.504,2.000,0.000,-180.000,-30.000
C00701=48.437,51.504,2.000,0.000,-180.000,-30.000
C00702=48.130,51.811,2.000,0.000,-180.000,-30.000
C00703=47.564,51.811,2.000,0.000,-180.000,-30.000
C00704=47.871,51.504,2.000,0.000,-180.000,-30.000
C00705=47.306,51.504,2.000,0.000,-180.000,-30.000
C00706=46.999,51.811,2.000,0.000,-180.000,-30.000
C00707=46.433,51.811,2.000,0.000,-180.000,-30.000
C00708=46.740,51.504,2.000,0.000,-180.000,-30.000
C00709=46.174,51.504,2.000,0.000,-180.000,-30.000
C00710=45.867,51.811,2.000,0.000,-180.000,-30.000
C00711=45.540,51.811,2.000,0.000,-180.000,-30.000
C00712=45.540,51.573,2.000,0.000,-180.000,-30.000
C00713=45.609,51.504,2.000,0.000,-180.000,-30.000
C00714=45.609,51.504,2.000,0.000,-180.000,-30.000
C00715=45.200,51.378,2.100,0.000,-180.000,-30.000
C00716=45.200,51.378,2.100,0.000,-180.000,-30.000
C00717=54.800,51.378,2.100,0.000,-180.000,-30.000
C00718=54.800,52.524,2.100,0.000,-180.000,-30.000
C00719=45.200,52.524,2.100,0.000,-180.000,-30.000
C00720=45.200,51.378,2.100,0.000,-180.000,-30.000
C00721=45.540,51.918,2.100,0.000,-180.000,-30.000
C00722=45.806,52.184,2.100,0.000,-180.000,-30.000
C00723=46.371,52.184,2.100,0.000,-180.000,-30.000
C00724=46.065,51.878,2.100,0.000,-180.000,-30.000
C00725=46.631,51.878,2.100,0.000,-180.000,-30.000
C00726=46.937,52.184,2.100,0.000,-180.000,-30.000
C00727=47.503,52.184,2.100,0.000,-180.000,-30.000
C00728=47.197,51.878,2.100,0.000,-180.000,-30.000
C00729=47.762,51.878,2.100,0.000,-180.000,-30.000
C00730=48.068,52.184,2.100,0.000,-180.000,-30.000
C00731=48.634,52.184,2.100,0.000,-180.000,-30.000
C00732=48.328,51.878,2.100,0.000,-180.000,-30.000
C00733=48.894,51.878,2.100,0.000,-180.000,-30.000
C00734=49.200,52.184,2.100,0.000,-180.000,-30.000
C00735=49.765,52.184,2.100,0.000,-180.000,-30.000
C00736=49.459,51.878,2.100,0.000,-180.000,-30.000
C00737=50.025,51.878,2.100,0.000,-180.000,-30.000
C00738=50.331,52.184,2.100,0.000,-180.000,-30.000
C00739=50.897,52.184,2.100,0.000,-180.000,-30.000
C00740=50.591,51.878,2.100,0.000,-180.000,-30.000
C00741=51.156,51.878,2.100,0.000,-180.000,-30.000
C00742=51.462,52.184,2.100,0.000,-180.000,-30.000
C00743=52.028,52.184,2.100,0.000,-180.000,-30.000
C00744=51.722,51.878,2.100,0.000,-180.000,-30.000
C00745=52.288,51.878,2.100,0.000,-180.000,-30.000
C00746=52.594,52.184,2.100,0.000,-180.000,-30.000
C00747=53.160,52.184,2.100,0.000,-180.000,-30.000
C00748=52.854,51.878,2.100,0.000,-180.000,-30.000
C00749=53.419,51.878,2.100,0.000,-180.000,-30.000
C00750=53.725,52.184,2.100,0.000,-180.000,-30.000
C00751=54.291,52.184,2.100,0.000,-180.000,-30.000
C00752=53.985,51.878,2.100,0.000,-180.000,-30.000
C00753=53.985,51.878,2.100,0.000,-180.000,-30.000
C00754=45.200,52.898,2.200,0.000,-180.000,-30.000
C00755=45.200,52.898,2.200,0.000,-180.000,-30.000
C00756=45.200,51.752,2.200,0.000,-180.000,-30.000
C00757=54.800,51.752,2.200,0.000,-180.000,-30.000
C00758=54.800,52.898,2.200,0.000,-180.000,-30.000
C00759=45.200,52.898,2.200,0.000,-180.000,-30.000
C00760=45.993,52.251,2.200,0.000,-180.000,-30.000
C00761=45.686,52.558,2.200,0.000,-180.000,-30.000
C00762=46.252,52.558,2.200,0.000,-180.000,-30.000
C00763=46.559,52.251,2.200,0.000,-180.000,-30.000
C00764=47.124,52.251,2.200,0.000,-180.000,-30.000
C00765=46.817,52.558,2.200,0.000,-180.000,-30.000
C00766=47.383,52.558,2.200,0.000,-180.000,-30.000
C00767=47.690,52.251,2.200,0.000,-180.000,-30.000
C00768=48.256,52.251,2.200,0.000,-180.000,-30.000
C00769=47.949,52.558,2.200,0.000,-180.000,-30.000
C00770=48.515,52.558,2.200,0.000,-180.000,-30.000
C00771=48.822,52.251,2.200,0.000,-180.000,-30.000
C00772=49.387,52.251,2.200,0.000,-180.000,-30.000
C00773=49.080,52.558,2.200,0.000,-180.000,-30.000
C00774=49.646,52.558,2.200,0.000,-180.000,-30.000
C00775=49.953,52.251,2.200,0.000,-180.000,-30.000
C00776=50.519,52.251,2.200,0.000,-180.000,-30.000
C00777=50.212,52.558,2.200,0.000,-180.000,-30.000
C00778=50.777,52.558,2.200,0.000,-180.000,-30.000
C00779=51.084,52.251,2.200,0.000,-180.000,-30.000
C00780=51.650,52.251,2.200,0.000,-180.000,-30.000
C00781=51.343,52.558,2.200,0.000,-180.000,-30.000
C00782=51.909,52.558,2.200,0.000,-180.000,-30.000
C00783=52.216,52.251,2.200,0.000,-180.000,-30.000
C00784=52.781,52.251,2.200,0.000,-180.000,-30.000
C00785=52.474,52.558,2.200,0.000,-180.000,-30.000
C00786=53.040,52.558,2.200,0.000,-180.000,-30.000
C00787=53.347,52.251,2.200,0.000,-180.000,-30.000
C00788=53.913,52.251,2.200,0.000,-180.000,-30.000
C00789=53.606,52.558,2.200,0.000,-180.000,-30.000
C00790=54.171,52.558,2.200,0.000,-180.000,-30.000
C00791=54.460,52.269,2.200,0.000,-180.000,-30.000
C00792=54.460,52.269,2.200,0.000,-180.000,-30.000
C00793=54.800,53.271,2.300,0.000,-180.000,-30.000
C00794=54.800,53.271,2.300,0.000,-180.000,-30.000
C00795=45.200,53.271,2.300,0.000,-180.000,-30.000
C00796=45.200,52.125,2.300,0.000,-180.000,-30.000
C00797=54.800,52.125,2.300,0.000,-180.000,-30.000
C00798=54.800,53.271,2.300,0.000,-180.000,-30.000
C00799=54.800,53.271,2.300,0.000,-180.000,-30.000
C00800=54.165,52.624,2.300,0.000,-180.000,-30.000
C00801=54.165,52.624,2.300,0.000,-180.000,-30.000
C00802=54.460,52.919,2.300,0.000,-180.000,-30.000
C00803=54.460,52.931,2.300,0.000,-180.000,-30.000
C00804=53.907,52.931,2.300,0.000,-180.000,-30.000
C00805=53.600,52.624,2.300,0.000,-180.000,-30.000
C00806=53.034,52.624,2.300,0.000,-180.000,-30.000
C00807=53.341,52.931,2.300,0.000,-180.000,-30.000
C00808=52.775,52.931,2.300,0.000,-180.000,-30.000
C00809=52.468,52.624,2.300,0.000,-180.000,-30.000
C00810=51.902,52.624,2.300,0.000,-180.000,-30.000
C00811=52.209,52.931,2.300,0.000,-180.000,-30.000
C00812=51.644,52.931,2.300,0.000,-180.000,-30.000
C00813=51.337,52.624,2.300,0.000,-180.000,-30.000
C00814=50.771,52.624,2.300,0.000,-180.000,-30.000
C00815=51.078,52.931,2.300,0.000,-180.000,-30.000
C00816=50.512,52.931,2.300,0.000,-180.000,-30.000
C00817=50.205,52.624,2.300,0.000,-180.000,-30.000
C00818=49.640,52.624,2.300,0.000,-180.000,-30.000
C00819=49.947,52.931,2.300,0.000,-180.000,-30.000
C00820=49.381,52.931,2.300,0.000,-180.000,-30.000
C00821=49.074,52.624,2.300,0.000,-180.000,-30.000
C00822=48.508,52.624,2.300,0.000,-180.000,-30.000
C00823=48.815,52.931,2.300,0.000,-180.000,-30.000
C00824=48.250,52.931,2.300,0.000,-180.000,-30.000
C00825=47.943,52.624,2.300,0.000,-180.000,-30.000
C00826=47.377,52.624,2.300,0.000,-180.000,-30.000
C00827=47.684,52.931,2.300,0.000,-180.000,-30.000
C00828=47.118,52.931,2.300,0.000,-180.000,-30.000
C00829=46.811,52.624,2.300,0.000,-180.000,-30.000
C00830=46.246,52.624,2.300,0.000,-180.000,-30.000
C00831=46.553,52.931,2.300,0.000,-180.000,-30.000
C00832=45.987,52.931,2.300,0.000,-180.000,-30.000
C00833=45.680,52.624,2.300,0.000,-180.000,-30.000
C00834=45.680,52.624,2.300,0.000,-180.000,-30.000
C00835=45.200,52.498,2.400,0.000,-180.000,-30.000
C00836=45.200,52.498,2.400,0.000,-180.000,-30.000
C00837=54.800,52.498,2.400,0.000,-180.000,-30.000
C00838=54.800,53.645,2.400,0.000,-180.000,-30.000
C00839=45.200,53.645,2.400,0.000,-180.000,-30.000
C00840=45.200,52.498,2.400,0.000,-180.000,-30.000
C00841=45.812,52.998,2.400,0.000,-180.000,-30.000
C00842=45.540,53.270,2.400,0.000,-180.000,-30.000
C00843=45.540,53.305,2.400,0.000,-180.000,-30.000
C00844=46.070,53.305,2.400,0.000,-180.000,-30.000
C00845=46.377,52.998,2.400,0.000,-180.000,-30.000
C00846=46.943,52.998,2.400,0.000,-180.000,-30.000
C00847=46.636,53.305,2.400,0.000,-180.000,-30.000
C00848=47.202,53.305,2.400,0.000,-180.000,-30.000
C00849=47.509,52.998,2.400,0.000,-180.000,-30.000
C00850=48.075,52.998,2.400,0.000,-180.000,-30.000
C00851=47.768,53.305,2.400,0.000,-180.000,-30.000
C00852=48.333,53.305,2.400,0.000,-180.000,-30.000
C00853=48.640,52.998,2.400,0.000,-180.000,-30.000
C00854=49.206,52.998,2.400,0.000,-180.000,-30.000
C00855=48.899,53.305,2.400,0.000,-180.000,-30.000
C00856=49.465,53.305,2.400,0.000,-180.000,-30.000
C00857=49.772,52.998,2.400,0.000,-180.000,-30.000
C00858=50.337,52.998,2.400,0.000,-180.000,-30.000
C00859=50.030,53.305,2.400,0.000,-180.000,-30.000
C00860=50.596,53.305,2.400,0.000,-180.000,-30.000
C00861=50.903,52.998,2.400,0.000,-180.000,-30.000
C00862=51.469,52.998,2.400,0.000,-180.000,-30.000
C00863=51.162,53.305,2.400,0.000,-180.000,-30.000
C00864=51.727,53.305,2.400,0.000,-180.000,-30.000
C00865=52.034,52.998,2.400,0.000,-180.000,-30.000
C00866=52.600,52.998,2.400,0.000,-180.000,-30.000
C00867=52.293,53.305,2.400,0.000,-180.000,-30.000
C00868=52.859,53.305,2.400,0.000,-180.000,-30.000
C00869=53.166,52.998,2.400,0.000,-180.000,-30.000
C00870=53.731,52.998,2.400,0.000,-180.000,-30.000
C00871=53.424,53.305,2.400,0.000,-180.000,-30.000
C00872=53.990,53.305,2.400,0.000,-180.000,-30.000
C00873=54.297,52.998,2.400,0.000,-180.000,-30.000
C00874=54.297,52.998,2.400,0.000,-180.000,-30.000
C00875=54.800,52.871,2.500,0.000,-180.000,-30.000
C00876=54.800,52.871,2.500,0.000,-180.000,-30.000
C00877=54.800,54.018,2.500,0.000,-180.000,-30.000
C00878=45.200,54.018,2.500,0.000,-180.000,-30.000
C00879=45.200,52.871,2.500,0.000,-180.000,-30.000
C00880=54.800,52.871,2.500,0.000,-180.000,-30.000
C00881=54.460,53.484,2.500,0.000,-180.000,-30.000
C00882=54.347,53.371,2.500,0.000,-180.000,-30.000
C00883=53.781,53.371,2.500,0.000,-180.000,-30.000
C00884=54.088,53.678,2.500,0.000,-180.000,-30.000
C00885=53.522,53.678,2.500,0.000,-180.000,-30.000
C00886=53.215,53.371,2.500,0.000,-180.000,-30.000
C00887=52.649,53.371,2.500,0.000,-180.000,-30.000
C00888=52.956,53.678,2.500,0.000,-180.000,-30.000
C00889=52.391,53.678,2.500,0.000,-180.000,-30.000
C00890=52.084,53.371,2.500,0.000,-180.000,-30.000
C00891=51.518,53.371,2.500,0.000,-180.000,-30.000
C00892=51.825,53.678,2.500,0.000,-180.000,-30.000
C00893=51.259,53.678,2.500,0.000,-180.000,-30.000
C00894=50.952,53.371,2.500,0.000,-180.000,-30.000
C00895=50.387,53.371,2.500,0.000,-180.000,-30.000
C00896=50.694,53.678,2.500,0.000,-180.000,-30.000
C00897=50.128,53.678,2.500,0.000,-180.000,-30.000
C00898=49.821,53.371,2.500,0.000,-180.000,-30.000
C00899=49.255,53.371,2.500,0.000,-180.000,-30.000
C00900=49.562,53.678,2.500,0.000,-180.000,-30.000
C00901=48.997,53.678,2.500,0.000,-180.000,-30.000
C00902=48.690,53.371,2.500,0.000,-180.000,-30.000
C00903=48.124,53.371,2.500,0.000,-180.000,-30.000
C00904=48.431,53.678,2.500,0.000,-180.000,-30.000
C00905=47.865,53.678,2.500,0.000,-180.000,-30.000
C00906=47.558,53.371,2.500,0.000,-180.000,-30.000
C00907=46.993,53.371,2.500,0.000,-180.000,-30.000
C00908=47.300,53.678,2.500,0.000,-180.000,-30.000
C00909=46.734,53.678,2.500,0.000,-180.000,-30.000
C00910=46.427,53.371,2.500,0.000,-180.000,-30.000
C00911=45.861,53.371,2.500,0.000,-180.000,-30.000
C00912=46.168,53.678,2.500,0.000,-180.000,-30.000
C00913=45.603,53.678,2.500,0.000,-180.000,-30.000
C00914=45.540,53.615,2.500,0.000,-180.000,-30.000
C00915=45.540,53.615,2.500,0.000,-180.000,-30.000
C00916=54.800,54.391,2.600,0.000,-180.000,-30.000
C00917=54.800,54.391,2.600,0.000,-180.000,-30.000
C00918=45.200,54.391,2.600,0.000,-180.000,-30.000
C00919=45.200,53.244,2.600,0.000,-180.000,-30.000
C00920=54.800,53.244,2.600,0.000,-180.000,-30.000
C00921=54.800,54.391,2.600,0.000,-180.000,-30.000
C00922=54.375,54.051,2.600,0.000,-180.000,-30.000
C00923=54.460,53.966,2.600,0.000,-180.000,-30.000
C00924=54.460,53.745,2.600,0.000,-180.000,-30.000
C00925=54.116,53.745,2.600,0.000,-180.000,-30.000
C00926=53.810,54.051,2.600,0.000,-180.000,-30.000
C00927=53.244,54.051,2.600,0.000,-180.000,-30.000
C00928=53.550,53.745,2.600,0.000,-180.000,-30.000
C00929=52.984,53.745,2.600,0.000,-180.000,-30.000
C00930=52.678,54.051,2.600,0.000,-180.000,-30.000
C00931=52.113,54.051,2.600,0.000,-180.000,-30.000
C00932=52.419,53.745,2.600,0.000,-180.000,-30.000
C00933=51.853,53.745,2.600,0.000,-180.000,-30.000
C00934=51.547,54.051,2.600,0.000,-180.000,-30.000
C00935=50.981,54.051,2.600,0.000,-180.000,-30.000
C00936=51.287,53.745,2.600,0.000,-180.000,-30.000
C00937=50.722,53.745,2.600,0.000,-180.000,-30.000
C00938=50.416,54.051,2.600,0.000,-180.000,-30.000
C00939=49.850,54.051,2.600,0.000,-180.000,-30.000
C00940=50.156,53.745,2.600,0.000,-180.000,-30.000
C00941=49.590,53.745,2.600,0.000,-180.000,-30.000
C00942=49.284,54.051,2.600,0.000,-180.000,-30.000
C00943=48.719,54.051,2.600,0.000,-180.000,-30.000
C00944=49.025,53.745,2.600,0.000,-180.000,-30.000
C00945=48.459,53.745,2.600,0.000,-180.000,-30.000
C00946=48.153,54.051,2.600,0.000,-180.000,-30.000
C00947=47.587,54.051,2.600,0.000,-180.000,-30.000
C00948=47.893,53.745,2.600,0.000,-180.000,-30.000
C00949=47.328,53.745,2.600,0.000,-180.000,-30.000
C00950=47.022,54.051,2.600,0.000,-180.000,-30.000
C00951=46.456,54.051,2.600,0.000,-180.000,-30.000
C00952=46.762,53.745,2.600,0.000,-180.000,-30.000
C00953=46.196,53.745,2.600,0.000,-180.000,-30.000
C00954=45.890,54.051,2.600,0.000,-180.000,-30.000
C00955=45.540,54.051,2.600,0.000,-180.000,-30.000
C00956=45.540,53.835,2.600,0.000,-180.000,-30.000
C00957=45.630,53.745,2.600,0.000,-180.000,-30.000
C00958=45.630,53.745,2.600,0.000,-180.000,-30.000
C00959=45.200,53.617,2.700,0.000,-180.000,-30.000
C00960=45.200,53.617,2.700,0.000,-180.000,-30.000
C00961=54.800,53.617,2.700,0.000,-180.000,-30.000
C00962=54.800,54.717,2.700,0.000,-180.000,-30.000
C00963=45.200,54.717,2.700,0.000,-180.000,-30.000
C00964=45.200,53.617,2.700,0.000,-180.000,-30.000
C00965=45.540,54.181,2.700,0.000,-180.000,-30.000
C00966=45.710,54.351,2.700,0.000,-180.000,-30.000
C00967=46.276,54.351,2.700,0.000,-180.000,-30.000
C00968=46.043,54.118,2.700,0.000,-180.000,-30.000
C00969=46.608,54.118,2.700,0.000,-180.000,-30.000
C00970=46.841,54.351,2.700,0.000,-180.000,-30.000
C00971=47.407,54.351,2.700,0.000,-180.000,-30.000
C00972=47.174,54.118,2.700,0.000,-180.000,-30.000
C00973=47.740,54.118,2.700,0.000,-180.000,-30.000
C00974=47.973,54.351,2.700,0.000,-180.000,-30.000
C00975=48.538,54.351,2.700,0.000,-180.000,-30.000
C00976=48.305,54.118,2.700,0.000,-180.000,-30.000
C00977=48.871,54.118,2.700,0.000,-180.000,-30.000
C00978=49.104,54.351,2.700,0.000,-180.000,-30.000
C00979=49.670,54.351,2.700,0.000,-180.000,-30.000
C00980=49.437,54.118,2.700,0.000,-180.000,-30.000
C00981=50.002,54.118,2.700,0.000,-180.000,-30.000
C00982=50.235,54.351,2.700,0.000,-180.000,-30.000
C00983=50.801,54.351,2.700,0.000,-180.000,-30.000
C00984=50.568,54.118,2.700,0.000,-180.000,-30.000
C00985=51.134,54.118,2.700,0.000,-180.000,-30.000
C00986=51.367,54.351,2.700,0.000,-180.000,-30.000
C00987=51.932,54.351,2.700,0.000,-180.000,-30.000
C00988=51.699,54.118,2.700,0.000,-180.000,-30.000
C00989=52.265,54.118,2.700,0.000,-180.000,-30.000
C00990=52.498,54.351,2.700,0.000,-180.000,-30.000
C00991=53.064,54.351,2.700,0.000,-180.000,-30.000
C00992=52.831,54.118,2.700,0.000,-180.000,-30.000
C00993=53.396,54.118,2.700,0.000,-180.000,-30.000
C00994=53.629,54.351,2.700,0.000,-180.000,-30.000
C00995=54.195,54.351,2.700,0.000,-180.000,-30.000
C00996=53.962,54.118,2.700,0.000,-180.000,-30.000
C00997=53.962,54.118,2.700,0.000,-180.000,-30.000
C00998=54.800,54.690,2.800,0.000,-180.000,-30.000
C00999=54.800,54.690,2.800,0.000,-180.000,-30.000
C01000=45.200,54.690,2.800,0.000,-180.000,-30.000
C01001=45.200,53.990,2.800,0.000,-180.000,-30.000
C01002=54.800,53.990,2.800,0.000,-180.000,-30.000
C01003=54.800,54.690,2.800,0.000,-180.000,-30.000
C01004=53.699,54.350,2.800,0.000,-180.000,-30.000
C01005=53.719,54.330,2.800,0.000,-180.000,-30.000
C01006=51.834,54.330,2.800,0.000,-180.000,-30.000
C01007=51.814,54.350,2.800,0.000,-180.000,-30.000
C01008=49.928,54.350,2.800,0.000,-180.000,-30.000
C01009=49.948,54.330,2.800,0.000,-180.000,-30.000
C01010=48.062,54.330,2.800,0.000,-180.000,-30.000
C01011=48.042,54.350,2.800,0.000,-180.000,-30.000
C01012=46.157,54.350,2.800,0.000,-180.000,-30.000
C01013=46.177,54.330,2.800,0.000,-180.000,-30.000
C01014=46.177,54.330,2.800,0.000,-180.000,-30.000
C01015=54.800,54.663,2.900,0.000,-180.000,-30.000
C01016=54.800,54.663,2.900,0.000,-180.000,-30.000
C01017=45.200,54.663,2.900,0.000,-180.000,-30.000
C01018=45.200,54.363,2.900,0.000,-180.000,-30.000
C01019=54.800,54.363,2.900,0.000,-180.000,-30.000
C01020=54.800,54.663,2.900,0.000,-180.000,-30.000
C01021=54.800,54.663,2.900,0.000,-180.000,-30.000
C01022=54.800,54.663,50.000,0.000,-180.000,-30.000
C01023=100.000,96.000,50.000,0.000,-180.000,-30.000
//INST
///ATTR SC,RW,RJ
////FRAME USER 1
///GROUP1 RB1
///LVARS 2,0,0,0,0,0,0,0
NOP
SET LB000 1
SET LB001 25
MOVJ C00000 VJ=17
' bead-prime
MOVL C00001 V=7 PL=LB000 ACC=LB001 DEC=LB001
MOVL C00002 V=25 PL=LB000 ACC=LB001 DEC=LB001
' rapid-dry
MOVL C00003 V=17 PL=LB000 ACC=LB001 DEC=LB001
MOVL C00004 V=25 PL=LB000 ACC=LB001 DEC=LB001
' bead-skirt/brim
MOVL C00005 V=13 PL=LB000 ACC=LB001 DEC=LB001
MOVL C00006 V=13 PL=LB000 ACC=LB001 DEC=LB001
MOVL C00007 V=13 PL=LB000 ACC=LB001 DEC=LB001
MOVL C00008 V=13 PL=LB000 ACC=LB001 DEC=LB001
' rapid-leaky
MOVL C00009 V=17 PL=LB000 ACC=LB001 DEC=LB001
' bead-skirt/brim
MOVL C00010 V=13 PL=LB000 ACC=LB001 DEC=LB001
MOVL C00011 V=13 PL=LB000 ACC=LB001 DEC=LB001
MOVL C00012 V=13 PL=LB000 ACC=LB001 DEC=LB001
MOVL C00013 V=13 PL=LB000 ACC=LB001 DEC=LB001
MOVL C00014 V=25 PL=LB000 ACC=LB001 DEC=LB001
' rapid-dry
MOVL C00015 V=17 PL=LB000 ACC=LB001 DEC=LB001
MOVL C00016 V=25 PL=LB000 ACC=LB001 DEC=LB001
' bead-perimeter_outer
MOVL C00017 V=20 PL=LB000 ACC=LB001 DEC=LB001
MOVL C00018 V=20 PL=LB000 ACC=LB001 DEC=LB001
MOVL C00019 V=20 PL=LB000 ACC=LB001 DEC=LB001
MOVL C00020 V=20 PL=LB000 ACC=LB001 DEC=LB001
MOVL C00021 V=25 PL=LB000 ACC=LB001 DEC=LB001
' rapid-dry
MOVL C00022 V=17 PL=LB000 ACC=LB001 DEC=LB001
MOVL C00023 V=25 PL=LB000 ACC=LB001 DEC=LB001
' bead-perimeter_outer
MOVL C00024 V=20 PL=LB000 ACC=LB001 DEC=LB001
MOVL C00025 V=20 PL=LB000 ACC=LB001 DEC=LB001
MOVL C00026 V=20 PL=LB000 ACC=LB001 DEC=LB001
MOVL C00027 V=20 PL=LB000 ACC=LB001 DEC=LB001
' rapid-leaky
MOVL C00028 V=17 PL=LB000 ACC=LB001 DEC=LB001
' bead-solid_infill
MOVL C00029 V=20 PL=LB000 ACC=LB001 DEC=LB001
MOVL C00030 V=20 PL=LB000 ACC=LB001 DEC=LB001
MOVL C00031 V=20 PL=LB000 ACC=LB001 DEC=LB001
MOVL C00032 V=20 PL=LB000 ACC=LB001 DEC=LB001
MOVL C00033 V=20 PL=LB000 ACC=LB001 DEC=LB001
MOVL C00034 V=20 PL=LB000 ACC=LB001 DEC=LB001
MOVL C00035 V=20 PL=LB000 ACC=LB001 DEC=LB001
MOVL C00036 V=20 PL=LB000 ACC=LB001 DEC=LB001
MOVL C00037 V=20 PL=LB000 ACC=LB001 DEC=LB001
MOVL C00038 V=20 PL=LB000 ACC=LB001 DEC=LB001
MOVL C00039 V=20 PL=LB000 ACC=LB001 DEC=LB001
MOVL C00040 V=20 PL=LB000 ACC=LB001 DEC=LB001
MOVL C00041 V=20 PL=LB000 ACC=LB001 DEC=LB001
MOVL C00042 V=20 PL=LB000 ACC=LB001 DEC=LB001
MOVL C00043 V=20 PL=LB000 ACC=LB001 DEC=LB001
MOVL C00044 V=20 PL=LB000 ACC=LB001 DEC=LB001
MOVL C00045 V=20 PL=LB000 ACC=LB001 DEC=LB001
MOVL C00046 V=20 PL=LB000 ACC=LB001 DEC=LB001
MOVL C00047 V=20 PL=LB000 ACC=LB001 DEC=LB001
MOVL C00048 V=20 PL=LB000 ACC=LB001 DEC=LB001
MOVL C00049 V=20 PL=LB000 ACC=LB001 DEC=LB001
MOVL C00050 V=20 PL=LB000 ACC=LB001 DEC=LB001
MOVL C00051 V=20 PL=LB000 ACC=LB001 DEC=LB001
MOVL C00052 V=20 PL=LB000 ACC=LB001 DEC=LB001
MOVL C00053 V=20 PL=LB000 ACC=LB001 DEC=LB001
MOVL C00054 V=20 PL=LB000 ACC=LB001 DEC=LB001
MOVL C00055 V=20 PL=LB000 ACC=LB001 DEC=LB001
MOVL C00056 V=20 PL=LB000 ACC=LB001 DEC=LB001
MOVL C00057 V=20 PL=LB000 ACC=LB001 DEC=LB001
MOVL C00058 V=20 PL=LB000 ACC=LB001 DEC=LB001
MOVL C00059 V=20 PL=LB000 ACC=LB001 DEC=LB001
MOVL C00060 V=25 PL=LB000 ACC=LB001 DEC=LB001
' rapid-dry
MOVL C00061 V=17 PL=LB000 ACC=LB001 DEC=LB001
MOVL C00062 V=25 PL=LB000 ACC=LB001 DEC=LB001
' bead-perimeter_outer
MOVL C00063 V=20 PL=LB000 ACC=LB001 DEC=LB001
MOVL C00064 V=20 PL=LB000 ACC=LB001 DEC=LB001
MOVL C00065 V=20 PL=LB000 ACC=LB001 DEC=LB001
MOVL C00066 V=20 PL=LB000 ACC=LB001 DEC=LB001
MOVL C00067 V=25 PL=LB000 ACC=LB001 DEC=LB001
' rapid-dry
MOVL C00068 V=17 PL=LB000 ACC=LB001 DEC=LB001
MOVL C00069 V=25 PL=LB000 ACC=LB001 DEC=LB001
' bead-solid_infill
MOVL C00070 V=20 PL=LB000 ACC=LB001 DEC=LB001
MOVL C00071 V=20 PL=LB000 ACC=LB001 DEC=LB001
MOVL C00072 V=20 PL=LB000 ACC=LB001 DEC=LB001
MOVL C00073 V=20 PL=LB000 ACC=LB001 DEC=LB001
MOVL C00074 V=20 PL=LB000 ACC=LB001 DEC=LB001
MOVL C00075 V=20 PL=LB000 ACC=LB001 DEC=LB001
MOVL C00076 V=20 PL=LB000 ACC=LB001 DEC=LB001
MOVL C00077 V=20 PL=LB000 ACC=LB001 DEC=LB001
MOVL C00078 V=20 PL=LB000 ACC=LB001 DEC=LB001
MOVL C00079 V=20 PL=LB000 ACC=LB001 DEC=LB001
MOVL C00080 V=20 PL=LB000 ACC=LB001 DEC=LB001
MOVL C00081 V=20 PL=LB000 ACC=LB001 DEC=LB001
MOVL C00082 V=20 PL=LB000 ACC=LB001 DEC=LB001
MOVL C00083 V=20 PL=LB000 ACC=LB001 DEC=LB001
MOVL C00084 V=20 PL=LB000 ACC=LB001 DEC=LB001
MOVL C00085 V=20 PL=LB000 ACC=LB001 DEC=LB001
MOVL C00086 V=20 PL=LB000 ACC=LB001 DEC=LB001
MOVL C00087 V=20 PL=LB000 ACC=LB001 DEC=LB001
MOVL C00088 V=20 PL=LB000 ACC=LB001 DEC=LB001
MOVL C00089 V=20 PL=LB000 ACC=LB001 DEC=LB001
MOVL C00090 V=20 PL=LB000 ACC=LB001 DEC=LB001
MOVL C00091 V=20 PL=LB000 ACC=LB001 DEC=LB001
MOVL C00092 V=20 PL=LB000 ACC=LB001 DEC=LB001
MOVL C00093 V=20 PL=LB000 ACC=LB001 DEC=LB001
MOVL C00094 V=20 PL=LB000 ACC=LB001 DEC=LB001
MOVL C00095 V=20 PL=LB000 ACC=LB001 DEC=LB001
MOVL C00096 V=20 PL=LB000 ACC=LB001 DEC=LB001
MOVL C00097 V=20 PL=LB000 ACC=LB001 DEC=LB001
MOVL C00098 V=20 PL=LB000 ACC=LB001 DEC=LB001
MOVL C00099 V=20 PL=LB000 ACC=LB001 DEC=LB001
MOVL C00100 V=20 PL=LB000 ACC=LB001 DEC=LB001
MOVL C00101 V=20 PL=LB000 ACC=LB001 DEC=LB001
MOVL C00102 V=25 PL=LB000 ACC=LB001 DEC=LB001
' rapid-leaky
MOVL C00103 V=17 PL=LB000 ACC=LB001 DEC=LB001
MOVL C00104 V=25 PL=LB000 ACC=LB001 DEC=LB001
' bead-perimeter_outer
MOVL C00105 V=20 PL=LB000 ACC=LB001 DEC=LB001
MOVL C00106 V=20 PL=LB000 ACC=LB001 DEC=LB001
MOVL C00107 V=20 PL=LB000 ACC=LB001 DEC=LB001
MOVL C00108 V=20 PL=LB000 ACC=LB001 DEC=LB001
' rapid-leaky
MOVL C00109 V=17 PL=LB000 ACC=LB001 DEC=LB001
' bead-solid_infill
MOVL C00110 V=20 PL=LB000 ACC=LB001 DEC=LB001
MOVL C00111 V=20 PL=LB000 ACC=LB001 DEC=LB001
MOVL C00112 V=20 PL=LB000 ACC=LB001 DEC=LB001
MOVL C00113 V=20 PL=LB000 ACC=LB001 DEC=LB001
MOVL C00114 V=20 PL=LB000 ACC=LB001 DEC=LB001
MOVL C00115 V=20 PL=LB000 ACC=LB001 DEC=LB001
MOVL C00116 V=20 PL=LB000 ACC=LB001 DEC=LB001
MOVL C00117 V=20 PL=LB000 ACC=LB001 DEC=LB001
MOVL C00118 V=20 PL=LB000 ACC=LB001 DEC=LB001
MOVL C00119 V=20 PL=LB000 ACC=LB001 DEC=LB001
MOVL C00120 V=20 PL=LB000 ACC=LB001 DEC=LB001
MOVL C00121 V=20 PL=LB000 ACC=LB001 DEC=LB001
MOVL C00122 V=20 PL=LB000 ACC=LB001 DEC=LB001
MOVL C00123 V=20 PL=LB000 ACC=LB001 DEC=LB001
MOVL C00124 V=20 PL=LB000 ACC=LB001 DEC=LB001
MOVL C00125 V=20 PL=LB000 ACC=LB001 DEC=LB001
MOVL C00126 V=20 PL=LB000 ACC=LB001 DEC=LB001
MOVL C00127 V=20 PL=LB000 ACC=LB001 DEC=LB001
MOVL C00128 V=20 PL=LB000 ACC=LB001 DEC=LB001
MOVL C00129 V=20 PL=LB000 ACC=LB001 DEC=LB001
MOVL C00130 V=20 PL=LB000 ACC=LB001 DEC=LB001
MOVL C00131 V=20 PL=LB000 ACC=LB001 DEC=LB001
MOVL C00132 V=20 PL=LB000 ACC=LB001 DEC=LB001
MOVL C00133 V=20 PL=LB000 ACC=LB001 DEC=LB001
MOVL C00134 V=20 PL=LB000 ACC=LB001 DEC=LB001
MOVL C00135 V=20 PL=LB000 ACC=LB001 DEC=LB001
MOVL C00136 V=20 PL=LB000 ACC=LB001 DEC=LB001
MOVL C00137 V=20 PL=LB000 ACC=LB001 DEC=LB001
MOVL C00138 V=20 PL=LB000 ACC=LB001 DEC=LB001
MOVL C00139 V=20 PL=LB000 ACC=LB001 DEC=LB001
MOVL C00140 V=20 PL=LB000 ACC=LB001 DEC=LB001
MOVL C00141 V=20 PL=LB000 ACC=LB001 DEC=LB001
MOVL C00142 V=25 PL=LB000 ACC=LB001 DEC=LB001
' rapid-leaky
MOVL C00143 V=17 PL=LB000 ACC=LB001 DEC=LB001
MOVL C00144 V=25 PL=LB000 ACC=LB001 DEC=LB001
' bead-perimeter_outer
MOVL C00145 V=20 PL=LB000 ACC=LB001 DEC=LB001
MOVL C00146 V=20 PL=LB000 ACC=LB001 DEC=LB001
MOVL C00147 V=20 PL=LB000 ACC=LB001 DEC=LB001
MOVL C00148 V=20 PL=LB000 ACC=LB001 DEC=LB001
' rapid-leaky
MOVL C00149 V=17 PL=LB000 ACC=LB001 DEC=LB001
' bead-solid_infill
MOVL C00150 V=20 PL=LB000 ACC=LB001 DEC=LB001
MOVL C00151 V=20 PL=LB000 ACC=LB001 DEC=LB001
MOVL C00152 V=20 PL=LB000 ACC=LB001 DEC=LB001
MOVL C00153 V=20 PL=LB000 ACC=LB001 DEC=LB001
MOVL C00154 V=20 PL=LB000 ACC=LB001 DEC=LB001
MOVL C00155 V=20 PL=LB000 ACC=LB001 DEC=LB001
MOVL C00156 V=20 PL=LB000 ACC=LB001 DEC=LB001
MOVL C00157 V=20 PL=LB000 ACC=LB001 DEC=LB001
MOVL C00158 V=20 PL=LB000 ACC=LB001 DEC=LB001
MOVL C00159 V=20 PL=LB000 ACC=LB001 DEC=LB001
MOVL C00160 V=20 PL=LB000 ACC=LB001 DEC=LB001
MOVL C00161 V=20 PL=LB000 ACC=LB001 DEC=LB001
MOVL C00162 V=20 PL=LB000 ACC=LB001 DEC=LB001
MOVL C00163 V=20 PL=LB000 ACC=LB001 DEC=LB001
MOVL C00164 V=20 PL=LB000 ACC=LB001 DEC=LB001
MOVL C00165 V=20 PL=LB000 ACC=LB001 DEC=LB001
MOVL C00166 V=20 PL=LB000 ACC=LB001 DEC=LB001
MOVL C00167 V=20 PL=LB000 ACC=LB001 DEC=LB001
MOVL C00168 V=20 PL=LB000 ACC=LB001 DEC=LB001
MOVL C00169 V=20 PL=LB000 ACC=LB001 DEC=LB001
MOVL C00170 V=20 PL=LB000 ACC=LB001 DEC=LB001
MOVL C00171 V=20 PL=LB000 ACC=LB001 DEC=LB001
MOVL C00172 V=20 PL=LB000 ACC=LB001 DEC=LB001
MOVL C00173 V=20 PL=LB000 ACC=LB001 DEC=LB001
MOVL C00174 V=20 PL=LB000 ACC=LB001 DEC=LB001
MOVL C00175 V=20 PL=LB000 ACC=LB001 DEC=LB001
MOVL C00176 V=20 PL=LB000 ACC=LB001 DEC=LB001
MOVL C00177 V=20 PL=LB000 ACC=LB001 DEC=LB001
MOVL C00178 V=20 PL=LB000 ACC=LB001 DEC=LB001
MOVL C00179 V=20 PL=LB000 ACC=LB001 DEC=LB001
MOVL C00180 V=20 PL=LB000 ACC=LB001 DEC=LB001
MOVL C00181 V=20 PL=LB000 ACC=LB001 DEC=LB001
MOVL C00182 V=20 PL=LB000 ACC=LB001 DEC=LB001
MOVL C00183 V=25 PL=LB000 ACC=LB001 DEC=LB001
' rapid-dry
MOVL C00184 V=17 PL=LB000 ACC=LB001 DEC=LB001
MOVL C00185 V=25 PL=LB000 ACC=LB001 DEC=LB001
' bead-perimeter_outer
MOVL C00186 V=20 PL=LB000 ACC=LB001 DEC=LB001
MOVL C00187 V=20 PL=LB000 ACC=LB001 DEC=LB001
MOVL C00188 V=20 PL=LB000 ACC=LB001 DEC=LB001
MOVL C00189 V=20 PL=LB000 ACC=LB001 DEC=LB001
' rapid-leaky
MOVL C00190 V=17 PL=LB000 ACC=LB001 DEC=LB001
' bead-solid_infill
MOVL C00191 V=20 PL=LB000 ACC=LB001 DEC=LB001
MOVL C00192 V=20 PL=LB000 ACC=LB001 DEC=LB001
MOVL C00193 V=20 PL=LB000 ACC=LB001 DEC=LB001
MOVL C00194 V=20 PL=LB000 ACC=LB001 DEC=LB001
MOVL C00195 V=20 PL=LB000 ACC=LB001 DEC=LB001
MOVL C00196 V=20 PL=LB000 ACC=LB001 DEC=LB001
MOVL C00197 V=20 PL=LB000 ACC=LB001 DEC=LB001
MOVL C00198 V=20 PL=LB000 ACC=LB001 DEC=LB001
MOVL C00199 V=20 PL=LB000 ACC=LB001 DEC=LB001
MOVL C00200 V=20 PL=LB000 ACC=LB001 DEC=LB001
MOVL C00201 V=20 PL=LB000 ACC=LB001 DEC=LB001
MOVL C00202 V=20 PL=LB000 ACC=LB001 DEC=LB001
MOVL C00203 V=20 PL=LB000 ACC=LB001 DEC=LB001
MOVL C00204 V=20 PL=LB000 ACC=LB001 DEC=LB001
MOVL C00205 V=20 PL=LB000 ACC=LB001 DEC=LB001
MOVL C00206 V=20 PL=LB000 ACC=LB001 DEC=LB001
MOVL C00207 V=20 PL=LB000 ACC=LB001 DEC=LB001
MOVL C00208 V=20 PL=LB000 ACC=LB001 DEC=LB001
MOVL C00209 V=20 PL=LB000 ACC=LB001 DEC=LB001
MOVL C00210 V=20 PL=LB000 ACC=LB001 DEC=LB001
MOVL C00211 V=20 PL=LB000 ACC=LB001 DEC=LB001
MOVL C00212 V=20 PL=LB000 ACC=LB001 DEC=LB001
MOVL C00213 V=20 PL=LB000 ACC=LB001 DEC=LB001
MOVL C00214 V=20 PL=LB000 ACC=LB001 DEC=LB001
MOVL C00215 V=20 PL=LB000 ACC=LB001 DEC=LB001
MOVL C00216 V=20 PL=LB000 ACC=LB001 DEC=LB001
MOVL C00217 V=20 PL=LB000 ACC=LB001 DEC=LB001
MOVL C00218 V=20 PL=LB000 ACC=LB001 DEC=LB001
MOVL C00219 V=20 PL=LB000 ACC=LB001 DEC=LB001
MOVL C00220 V=20 PL=LB000 ACC=LB001 DEC=LB001
MOVL C00221 V=20 PL=LB000 ACC=LB001 DEC=LB001
MOVL C00222 V=20 PL=LB000 ACC=LB001 DEC=LB001
MOVL C00223 V=20 PL=LB000 ACC=LB001 DEC=LB001
MOVL C00224 V=20 PL=LB000 ACC=LB001 DEC=LB001
MOVL C00225 V=20 PL=LB000 ACC=LB001 DEC=LB001
MOVL C00226 V=25 PL=LB000 ACC=LB001 DEC=LB001
' rapid-leaky
MOVL C00227 V=17 PL=LB000 ACC=LB001 DEC=LB001
MOVL C00228 V=25 PL=LB000 ACC=LB001 DEC=LB001
' bead-perimeter_outer
MOVL C00229 V=20 PL=LB000 ACC=LB001 DEC=LB001
MOVL C00230 V=20 PL=LB000 ACC=LB001 DEC=LB001
MOVL C00231 V=20 PL=LB000 ACC=LB001 DEC=LB001
MOVL C00232 V=20 PL=LB000 ACC=LB001 DEC=LB001
' rapid-leaky
MOVL C00233 V=17 PL=LB000 ACC=LB001 DEC=LB001
' bead-solid_infill
MOVL C00234 V=20 PL=LB000 ACC=LB001 DEC=LB001
MOVL C00235 V=20 PL=LB000 ACC=LB001 DEC=LB001
MOVL C00236 V=20 PL=LB000 ACC=LB001 DEC=LB001
MOVL C00237 V=20 PL=LB000 ACC=LB001 DEC=LB001
MOVL C00238 V=20 PL=LB000 ACC=LB001 DEC=LB001
MOVL C00239 V=20 PL=LB000 ACC=LB001 DEC=LB001
MOVL C00240 V=20 PL=LB000 ACC=LB001 DEC=LB001
MOVL C00241 V=20 PL=LB000 ACC=LB001 DEC=LB001
MOVL C00242 V=20 PL=LB000 ACC=LB001 DEC=LB001
MOVL C00243 V=20 PL=LB000 ACC=LB001 DEC=LB001
MOVL C00244 V=20 PL=LB000 ACC=LB001 DEC=LB001
MOVL C00245 V=20 PL=LB000 ACC=LB001 DEC=LB001
MOVL C00246 V=20 PL=LB000 ACC=LB001 DEC=LB001
MOVL C00247 V=20 PL=LB000 ACC=LB001 DEC=LB001
MOVL C00248 V=20 PL=LB000 ACC=LB001 DEC=LB001
MOVL C00249 V=20 PL=LB000 ACC=LB001 DEC=LB001
MOVL C00250 V=20 PL=LB000 ACC=LB001 DEC=LB001
MOVL C00251 V=20 PL=LB000 ACC=LB001 DEC=LB001
MOVL C00252 V=20 PL=LB000 ACC=LB001 DEC=LB001
MOVL C00253 V=20 PL=LB000 ACC=LB001 DEC=LB001
MOVL C00254 V=20 PL=LB000 ACC=LB001 DEC=LB001
MOVL C00255 V=20 PL=LB000 ACC=LB001 DEC=LB001
MOVL C00256 V=20 PL=LB000 ACC=LB001 DEC=LB001
MOVL C00257 V=20 PL=LB000 ACC=LB001 DEC=LB001
MOVL C00258 V=20 PL=LB000 ACC=LB001 DEC=LB001
MOVL C00259 V=20 PL=LB000 ACC=LB001 DEC=LB001
MOVL C00260 V=20 PL=LB000 ACC=LB001 DEC=LB001
MOVL C00261 V=20 PL=LB000 ACC=LB001 DEC=LB001
MOVL C00262 V=20 PL=LB000 ACC=LB001 DEC=LB001
MOVL C00263 V=20 PL=LB000 ACC=LB001 DEC=LB001
MOVL C00264 V=20 PL=LB000 ACC=LB001 DEC=LB001
MOVL C00265 V=25 PL=LB000 ACC=LB001 DEC=LB001
' rapid-dry
MOVL C00266 V=17 PL=LB000 ACC=LB001 DEC=LB001
MOVL C00267 V=25 PL=LB000 ACC=LB001 DEC=LB001
' bead-perimeter_outer
MOVL C00268 V=20 PL=LB000 ACC=LB001 DEC=LB001
MOVL C00269 V=20 PL=LB000 ACC=LB001 DEC=LB001
MOVL C00270 V=20 PL=LB000 ACC=LB001 DEC=LB001
MOVL C00271 V=20 PL=LB000 ACC=LB001 DEC=LB001
' rapid-leaky
MOVL C00272 V=17 PL=LB000 ACC=LB001 DEC=LB001
' bead-solid_infill
MOVL C00273 V=20 PL=LB000 ACC=LB001 DEC=LB001
MOVL C00274 V=20 PL=LB000 ACC=LB001 DEC=LB001
MOVL C00275 V=20 PL=LB000 ACC=LB001 DEC=LB001
MOVL C00276 V=20 PL=LB000 ACC=LB001 DEC=LB001
MOVL C00277 V=20 PL=LB000 ACC=LB001 DEC=LB001
MOVL C00278 V=20 PL=LB000 ACC=LB001 DEC=LB001
MOVL C00279 V=20 PL=LB000 ACC=LB001 DEC=LB001
MOVL C00280 V=20 PL=LB000 ACC=LB001 DEC=LB001
MOVL C00281 V=20 PL=LB000 ACC=LB001 DEC=LB001
MOVL C00282 V=20 PL=LB000 ACC=LB001 DEC=LB001
MOVL C00283 V=20 PL=LB000 ACC=LB001 DEC=LB001
MOVL C00284 V=20 PL=LB000 ACC=LB001 DEC=LB001
MOVL C00285 V=20 PL=LB000 ACC=LB001 DEC=LB001
MOVL C00286 V=20 PL=LB000 ACC=LB001 DEC=LB001
MOVL C00287 V=20 PL=LB000 ACC=LB001 DEC=LB001
MOVL C00288 V=20 PL=LB000 ACC=LB001 DEC=LB001
MOVL C00289 V=20 PL=LB000 ACC=LB001 DEC=LB001
MOVL C00290 V=20 PL=LB000 ACC=LB001 DEC=LB001
MOVL C00291 V=20 PL=LB000 ACC=LB001 DEC=LB001
MOVL C00292 V=20 PL=LB000 ACC=LB001 DEC=LB001
MOVL C00293 V=20 PL=LB000 ACC=LB001 DEC=LB001
MOVL C00294 V=20 PL=LB000 ACC=LB001 DEC=LB001
MOVL C00295 V=20 PL=LB000 ACC=LB001 DEC=LB001
MOVL C00296 V=20 PL=LB000 ACC=LB001 DEC=LB001
MOVL C00297 V=20 PL=LB000 ACC=LB001 DEC=LB001
MOVL C00298 V=20 PL=LB000 ACC=LB001 DEC=LB001
MOVL C00299 V=20 PL=LB000 ACC=LB001 DEC=LB001
MOVL C00300 V=20 PL=LB000 ACC=LB001 DEC=LB001
MOVL C00301 V=20 PL=LB000 ACC=LB001 DEC=LB001
MOVL C00302 V=20 PL=LB000 ACC=LB001 DEC=LB001
MOVL C00303 V=20 PL=LB000 ACC=LB001 DEC=LB001
MOVL C00304 V=25 PL=LB000 ACC=LB001 DEC=LB001
' rapid-dry
MOVL C00305 V=17 PL=LB000 ACC=LB001 DEC=LB001
MOVL C00306 V=25 PL=LB000 ACC=LB001 DEC=LB001
' bead-perimeter_outer
MOVL C00307 V=20 PL=LB000 ACC=LB001 DEC=LB001
MOVL C00308 V=20 PL=LB000 ACC=LB001 DEC=LB001
MOVL C00309 V=20 PL=LB000 ACC=LB001 DEC=LB001
MOVL C00310 V=20 PL=LB000 ACC=LB001 DEC=LB001
MOVL C00311 V=25 PL=LB000 ACC=LB001 DEC=LB001
' rapid-dry
MOVL C00312 V=17 PL=LB000 ACC=LB001 DEC=LB001
MOVL C00313 V=25 PL=LB000 ACC=LB001 DEC=LB001
' bead-solid_infill
MOVL C00314 V=20 PL=LB000 ACC=LB001 DEC=LB001
MOVL C00315 V=20 PL=LB000 ACC=LB001 DEC=LB001
MOVL C00316 V=20 PL=LB000 ACC=LB001 DEC=LB001
MOVL C00317 V=20 PL=LB000 ACC=LB001 DEC=LB001
MOVL C00318 V=20 PL=LB000 ACC=LB001 DEC=LB001
MOVL C00319 V=20 PL=LB000 ACC=LB001 DEC=LB001
MOVL C00320 V=20 PL=LB000 ACC=LB001 DEC=LB001
MOVL C00321 V=20 PL=LB000 ACC=LB001 DEC=LB001
MOVL C00322 V=20 PL=LB000 ACC=LB001 DEC=LB001
MOVL C00323 V=20 PL=LB000 ACC=LB001 DEC=LB001
MOVL C00324 V=20 PL=LB000 ACC=LB001 DEC=LB001
MOVL C00325 V=20 PL=LB000 ACC=LB001 DEC=LB001
MOVL C00326 V=20 PL=LB000 ACC=LB001 DEC=LB001
MOVL C00327 V=20 PL=LB000 ACC=LB001 DEC=LB001
MOVL C00328 V=20 PL=LB000 ACC=LB001 DEC=LB001
MOVL C00329 V=20 PL=LB000 ACC=LB001 DEC=LB001
MOVL C00330 V=20 PL=LB000 ACC=LB001 DEC=LB001
MOVL C00331 V=20 PL=LB000 ACC=LB001 DEC=LB001
MOVL C00332 V=20 PL=LB000 ACC=LB001 DEC=LB001
MOVL C00333 V=20 PL=LB000 ACC=LB001 DEC=LB001
MOVL C00334 V=20 PL=LB000 ACC=LB001 DEC=LB001
MOVL C00335 V=20 PL=LB000 ACC=LB001 DEC=LB001
MOVL C00336 V=20 PL=LB000 ACC=LB001 DEC=LB001
MOVL C00337 V=20 PL=LB000 ACC=LB001 DEC=LB001
MOVL C00338 V=20 PL=LB000 ACC=LB001 DEC=LB001
MOVL C00339 V=20 PL=LB000 ACC=LB001 DEC=LB001
MOVL C00340 V=20 PL=LB000 ACC=LB001 DEC=LB001
MOVL C00341 V=20 PL=LB000 ACC=LB001 DEC=LB001
MOVL C00342 V=20 PL=LB000 ACC=LB001 DEC=LB001
MOVL C00343 V=20 PL=LB000 ACC=LB001 DEC=LB001
MOVL C00344 V=20 PL=LB000 ACC=LB001 DEC=LB001
MOVL C00345 V=20 PL=LB000 ACC=LB001 DEC=LB001
MOVL C00346 V=25 PL=LB000 ACC=LB001 DEC=LB001
' rapid-leaky
MOVL C00347 V=17 PL=LB000 ACC=LB001 DEC=LB001
MOVL C00348 V=25 PL=LB000 ACC=LB001 DEC=LB001
' bead-perimeter_outer
MOVL C00349 V=20 PL=LB000 ACC=LB001 DEC=LB001
MOVL C00350 V=20 PL=LB000 ACC=LB001 DEC=LB001
MOVL C00351 V=20 PL=LB000 ACC=LB001 DEC=LB001
MOVL C00352 V=20 PL=LB000 ACC=LB001 DEC=LB001
MOVL C00353 V=25 PL=LB000 ACC=LB001 DEC=LB001
' rapid-dry
MOVL C00354 V=17 PL=LB000 ACC=LB001 DEC=LB001
MOVL C00355 V=25 PL=LB000 ACC=LB001 DEC=LB001
' bead-solid_infill
MOVL C00356 V=20 PL=LB000 ACC=LB001 DEC=LB001
MOVL C00357 V=20 PL=LB000 ACC=LB001 DEC=LB001
MOVL C00358 V=20 PL=LB000 ACC=LB001 DEC=LB001
MOVL C00359 V=20 PL=LB000 ACC=LB001 DEC=LB001
MOVL C00360 V=20 PL=LB000 ACC=LB001 DEC=LB001
MOVL C00361 V=20 PL=LB000 ACC=LB001 DEC=LB001
MOVL C00362 V=20 PL=LB000 ACC=LB001 DEC=LB001
MOVL C00363 V=20 PL=LB000 ACC=LB001 DEC=LB001
MOVL C00364 V=20 PL=LB000 ACC=LB001 DEC=LB001
MOVL C00365 V=20 PL=LB000 ACC=LB001 DEC=LB001
MOVL C00366 V=20 PL=LB000 ACC=LB001 DEC=LB001
MOVL C00367 V=20 PL=LB000 ACC=LB001 DEC=LB001
MOVL C00368 V=20 PL=LB000 ACC=LB001 DEC=LB001
MOVL C00369 V=20 PL=LB000 ACC=LB001 DEC=LB001
MOVL C00370 V=20 PL=LB000 ACC=LB001 DEC=LB001
MOVL C00371 V=20 PL=LB000 ACC=LB001 DEC=LB001
MOVL C00372 V=20 PL=LB000 ACC=LB001 DEC=LB001
MOVL C00373 V=20 PL=LB000 ACC=LB001 DEC=LB001
MOVL C00374 V=20 PL=LB000 ACC=LB001 DEC=LB001
MOVL C00375 V=20 PL=LB000 ACC=LB001 DEC=LB001
MOVL C00376 V=20 PL=LB000 ACC=LB001 DEC=LB001
MOVL C00377 V=20 PL=LB000 ACC=LB001 DEC=LB001
MOVL C00378 V=20 PL=LB000 ACC=LB001 DEC=LB001
MOVL C00379 V=20 PL=LB000 ACC=LB001 DEC=LB001
MOVL C00380 V=20 PL=LB000 ACC=LB001 DEC=LB001
MOVL C00381 V=20 PL=LB000 ACC=LB001 DEC=LB001
MOVL C00382 V=20 PL=LB000 ACC=LB001 DEC=LB001
MOVL C00383 V=20 PL=LB000 ACC=LB001 DEC=LB001
MOVL C00384 V=20 PL=LB000 ACC=LB001 DEC=LB001
MOVL C00385 V=20 PL=LB000 ACC=LB001 DEC=LB001
MOVL C00386 V=20 PL=LB000 ACC=LB001 DEC=LB001
MOVL C00387 V=20 PL=LB000 ACC=LB001 DEC=LB001
MOVL C00388 V=25 PL=LB000 ACC=LB001 DEC=LB001
' rapid-dry
MOVL C00389 V=17 PL=LB000 ACC=LB001 DEC=LB001
MOVL C00390 V=25 PL=LB000 ACC=LB001 DEC=LB001
' bead-perimeter_outer
MOVL C00391 V=20 PL=LB000 ACC=LB001 DEC=LB001
MOVL C00392 V=20 PL=LB000 ACC=LB001 DEC=LB001
MOVL C00393 V=20 PL=LB000 ACC=LB001 DEC=LB001
MOVL C00394 V=20 PL=LB000 ACC=LB001 DEC=LB001
' rapid-leaky
MOVL C00395 V=17 PL=LB000 ACC=LB001 DEC=LB001
' bead-solid_infill
MOVL C00396 V=20 PL=LB000 ACC=LB001 DEC=LB001
MOVL C00397 V=20 PL=LB000 ACC=LB001 DEC=LB001
MOVL C00398 V=20 PL=LB000 ACC=LB001 DEC=LB001
MOVL C00399 V=20 PL=LB000 ACC=LB001 DEC=LB001
MOVL C00400 V=20 PL=LB000 ACC=LB001 DEC=LB001
MOVL C00401 V=20 PL=LB000 ACC=LB001 DEC=LB001
MOVL C00402 V=20 PL=LB000 ACC=LB001 DEC=LB001
MOVL C00403 V=20 PL=LB000 ACC=LB001 DEC=LB001
MOVL C00404 V=20 PL=LB000 ACC=LB001 DEC=LB001
MOVL C00405 V=20 PL=LB000 ACC=LB001 DEC=LB001
MOVL C00406 V=20 PL=LB000 ACC=LB001 DEC=LB001
MOVL C00407 V=20 PL=LB000 ACC=LB001 DEC=LB001
MOVL C00408 V=20 PL=LB000 ACC=LB001 DEC=LB001
MOVL C00409 V=20 PL=LB000 ACC=LB001 DEC=LB001
MOVL C00410 V=20 PL=LB000 ACC=LB001 DEC=LB001
MOVL C00411 V=20 PL=LB000 ACC=LB001 DEC=LB001
MOVL C00412 V=20 PL=LB000 ACC=LB001 DEC=LB001
MOVL C00413 V=20 PL=LB000 ACC=LB001 DEC=LB001
MOVL C00414 V=20 PL=LB000 ACC=LB001 DEC=LB001
MOVL C00415 V=20 PL=LB000 ACC=LB001 DEC=LB001
MOVL C00416 V=20 PL=LB000 ACC=LB001 DEC=LB001
MOVL C00417 V=20 PL=LB000 ACC=LB001 DEC=LB001
MOVL C00418 V=20 PL=LB000 ACC=LB001 DEC=LB001
MOVL C00419 V=20 PL=LB000 ACC=LB001 DEC=LB001
MOVL C00420 V=20 PL=LB000 ACC=LB001 DEC=LB001
MOVL C00421 V=20 PL=LB000 ACC=LB001 DEC=LB001
MOVL C00422 V=20 PL=LB000 ACC=LB001 DEC=LB001
MOVL C00423 V=20 PL=LB000 ACC=LB001 DEC=LB001
MOVL C00424 V=20 PL=LB000 ACC=LB001 DEC=LB001
MOVL C00425 V=20 PL=LB000 ACC=LB001 DEC=LB001
MOVL C00426 V=20 PL=LB000 ACC=LB001 DEC=LB001
MOVL C00427 V=20 PL=LB000 ACC=LB001 DEC=LB001
MOVL C00428 V=20 PL=LB000 ACC=LB001 DEC=LB001
MOVL C00429 V=25 PL=LB000 ACC=LB001 DEC=LB001
' rapid-leaky
MOVL C00430 V=17 PL=LB000 ACC=LB001 DEC=LB001
MOVL C00431 V=25 PL=LB000 ACC=LB001 DEC=LB001
' bead-perimeter_outer
MOVL C00432 V=20 PL=LB000 ACC=LB001 DEC=LB001
MOVL C00433 V=20 PL=LB000 ACC=LB001 DEC=LB001
MOVL C00434 V=20 PL=LB000 ACC=LB001 DEC=LB001
MOVL C00435 V=20 PL=LB000 ACC=LB001 DEC=LB001
' rapid-leaky
MOVL C00436 V=17 PL=LB000 ACC=LB001 DEC=LB001
' bead-solid_infill
MOVL C00437 V=20 PL=LB000 ACC=LB001 DEC=LB001
MOVL C00438 V=20 PL=LB000 ACC=LB001 DEC=LB001
MOVL C00439 V=20 PL=LB000 ACC=LB001 DEC=LB001
MOVL C00440 V=20 PL=LB000 ACC=LB001 DEC=LB001
MOVL C00441 V=20 PL=LB000 ACC=LB001 DEC=LB001
MOVL C00442 V=20 PL=LB000 ACC=LB001 DEC=LB001
MOVL C00443 V=20 PL=LB000 ACC=LB001 DEC=LB001
MOVL C00444 V=20 PL=LB000 ACC=LB001 DEC=LB001
MOVL C00445 V=20 PL=LB000 ACC=LB001 DEC=LB001
MOVL C00446 V=20 PL=LB000 ACC=LB001 DEC=LB001
MOVL C00447 V=20 PL=LB000 ACC=LB001 DEC=LB001
MOVL C00448 V=20 PL=LB000 ACC=LB001 DEC=LB001
MOVL C00449 V=20 PL=LB000 ACC=LB001 DEC=LB001
MOVL C00450 V=20 PL=LB000 ACC=LB001 DEC=LB001
MOVL C00451 V=20 PL=LB000 ACC=LB001 DEC=LB001
MOVL C00452 V=20 PL=LB000 ACC=LB001 DEC=LB001
MOVL C00453 V=20 PL=LB000 ACC=LB001 DEC=LB001
MOVL C00454 V=20 PL=LB000 ACC=LB001 DEC=LB001
MOVL C00455 V=20 PL=LB000 ACC=LB001 DEC=LB001
MOVL C00456 V=20 PL=LB000 ACC=LB001 DEC=LB001
MOVL C00457 V=20 PL=LB000 ACC=LB001 DEC=LB001
MOVL C00458 V=20 PL=LB000 ACC=LB001 DEC=LB001
MOVL C00459 V=20 PL=LB000 ACC=LB001 DEC=LB001
MOVL C00460 V=20 PL=LB000 ACC=LB001 DEC=LB001
MOVL C00461 V=20 PL=LB000 ACC=LB001 DEC=LB001
MOVL C00462 V=20 PL=LB000 ACC=LB001 DEC=LB001
MOVL C00463 V=20 PL=LB000 ACC=LB001 DEC=LB001
MOVL C00464 V=20 PL=LB000 ACC=LB001 DEC=LB001
MOVL C00465 V=20 PL=LB000 ACC=LB001 DEC=LB001
MOVL C00466 V=20 PL=LB000 ACC=LB001 DEC=LB001
MOVL C00467 V=20 PL=LB000 ACC=LB001 DEC=LB001
MOVL C00468 V=20 PL=LB000 ACC=LB001 DEC=LB001
MOVL C00469 V=20 PL=LB000 ACC=LB001 DEC=LB001
MOVL C00470 V=20 PL=LB000 ACC=LB001 DEC=LB001
MOVL C00471 V=20 PL=LB000 ACC=LB001 DEC=LB001
MOVL C00472 V=25 PL=LB000 ACC=LB001 DEC=LB001
' rapid-dry
MOVL C00473 V=17 PL=LB000 ACC=LB001 DEC=LB001
MOVL C00474 V=25 PL=LB000 ACC=LB001 DEC=LB001
' bead-perimeter_outer
MOVL C00475 V=20 PL=LB000 ACC=LB001 DEC=LB001
MOVL C00476 V=20 PL=LB000 ACC=LB001 DEC=LB001
MOVL C00477 V=20 PL=LB000 ACC=LB001 DEC=LB001
MOVL C00478 V=20 PL=LB000 ACC=LB001 DEC=LB001
' rapid-leaky
MOVL C00479 V=17 PL=LB000 ACC=LB001 DEC=LB001
' bead-solid_infill
MOVL C00480 V=20 PL=LB000 ACC=LB001 DEC=LB001
MOVL C00481 V=20 PL=LB000 ACC=LB001 DEC=LB001
MOVL C00482 V=20 PL=LB000 ACC=LB001 DEC=LB001
MOVL C00483 V=20 PL=LB000 ACC=LB001 DEC=LB001
MOVL C00484 V=20 PL=LB000 ACC=LB001 DEC=LB001
MOVL C00485 V=20 PL=LB000 ACC=LB001 DEC=LB001
MOVL C00486 V=20 PL=LB000 ACC=LB001 DEC=LB001
MOVL C00487 V=20 PL=LB000 ACC=LB001 DEC=LB001
MOVL C00488 V=20 PL=LB000 ACC=LB001 DEC=LB001
MOVL C00489 V=20 PL=LB000 ACC=LB001 DEC=LB001
MOVL C00490 V=20 PL=LB000 ACC=LB001 DEC=LB001
MOVL C00491 V=20 PL=LB000 ACC=LB001 DEC=LB001
MOVL C00492 V=20 PL=LB000 ACC=LB001 DEC=LB001
MOVL C00493 V=20 PL=LB000 ACC=LB001 DEC=LB001
MOVL C00494 V=20 PL=LB000 ACC=LB001 DEC=LB001
MOVL C00495 V=20 PL=LB000 ACC=LB001 DEC=LB001
MOVL C00496 V=20 PL=LB000 ACC=LB001 DEC=LB001
MOVL C00497 V=20 PL=LB000 ACC=LB001 DEC=LB001
MOVL C00498 V=20 PL=LB000 ACC=LB001 DEC=LB001
MOVL C00499 V=20 PL=LB000 ACC=LB001 DEC=LB001
MOVL C00500 V=20 PL=LB000 ACC=LB001 DEC=LB001
MOVL C00501 V=20 PL=LB000 ACC=LB001 DEC=LB001
MOVL C00502 V=20 PL=LB000 ACC=LB001 DEC=LB001
MOVL C00503 V=20 PL=LB000 ACC=LB001 DEC=LB001
MOVL C00504 V=20 PL=LB000 ACC=LB001 DEC=LB001
MOVL C00505 V=20 PL=LB000 ACC=LB001 DEC=LB001
MOVL C00506 V=20 PL=LB000 ACC=LB001 DEC=LB001
MOVL C00507 V=20 PL=LB000 ACC=LB001 DEC=LB001
MOVL C00508 V=20 PL=LB000 ACC=LB001 DEC=LB001
MOVL C00509 V=20 PL=LB000 ACC=LB001 DEC=LB001
MOVL C00510 V=20 PL=LB000 ACC=LB001 DEC=LB001
MOVL C00511 V=25 PL=LB000 ACC=LB001 DEC=LB001
' rapid-dry
MOVL C00512 V=17 PL=LB000 ACC=LB001 DEC=LB001
MOVL C00513 V=25 PL=LB000 ACC=LB001 DEC=LB001
' bead-perimeter_outer
MOVL C00514 V=20 PL=LB000 ACC=LB001 DEC=LB001
MOVL C00515 V=20 PL=LB000 ACC=LB001 DEC=LB001
MOVL C00516 V=20 PL=LB000 ACC=LB001 DEC=LB001
MOVL C00517 V=20 PL=LB000 ACC=LB001 DEC=LB001
' rapid-leaky
MOVL C00518 V=17 PL=LB000 ACC=LB001 DEC=LB001
' bead-solid_infill
MOVL C00519 V=20 PL=LB000 ACC=LB001 DEC=LB001
MOVL C00520 V=20 PL=LB000 ACC=LB001 DEC=LB001
MOVL C00521 V=20 PL=LB000 ACC=LB001 DEC=LB001
MOVL C00522 V=20 PL=LB000 ACC=LB001 DEC=LB001
MOVL C00523 V=20 PL=LB000 ACC=LB001 DEC=LB001
MOVL C00524 V=20 PL=LB000 ACC=LB001 DEC=LB001
MOVL C00525 V=20 PL=LB000 ACC=LB001 DEC=LB001
MOVL C00526 V=20 PL=LB000 ACC=LB001 DEC=LB001
MOVL C00527 V=20 PL=LB000 ACC=LB001 DEC=LB001
MOVL C00528 V=20 PL=LB000 ACC=LB001 DEC=LB001
MOVL C00529 V=20 PL=LB000 ACC=LB001 DEC=LB001
MOVL C00530 V=20 PL=LB000 ACC=LB001 DEC=LB001
MOVL C00531 V=20 PL=LB000 ACC=LB001 DEC=LB001
MOVL C00532 V=20 PL=LB000 ACC=LB001 DEC=LB001
MOVL C00533 V=20 PL=LB000 ACC=LB001 DEC=LB001
MOVL C00534 V=20 PL=LB000 ACC=LB001 DEC=LB001
MOVL C00535 V=20 PL=LB000 ACC=LB001 DEC=LB001
MOVL C00536 V=20 PL=LB000 ACC=LB001 DEC=LB001
MOVL C00537 V=20 PL=LB000 ACC=LB001 DEC=LB001
MOVL C00538 V=20 PL=LB000 ACC=LB001 DEC=LB001
MOVL C00539 V=20 PL=LB000 ACC=LB001 DEC=LB001
MOVL C00540 V=20 PL=LB000 ACC=LB001 DEC=LB001
MOVL C00541 V=20 PL=LB000 ACC=LB001 DEC=LB001
MOVL C00542 V=20 PL=LB000 ACC=LB001 DEC=LB001
MOVL C00543 V=20 PL=LB000 ACC=LB001 DEC=LB001
MOVL C00544 V=20 PL=LB000 ACC=LB001 DEC=LB001
MOVL C00545 V=20 PL=LB000 ACC=LB001 DEC=LB001
MOVL C00546 V=20 PL=LB000 ACC=LB001 DEC=LB001
MOVL C00547 V=20 PL=LB000 ACC=LB001 DEC=LB001
MOVL C00548 V=20 PL=LB000 ACC=LB001 DEC=LB001
MOVL C00549 V=20 PL=LB000 ACC=LB001 DEC=LB001
MOVL C00550 V=25 PL=LB000 ACC=LB001 DEC=LB001
' rapid-leaky
MOVL C00551 V=17 PL=LB000 ACC=LB001 DEC=LB001
MOVL C00552 V=25 PL=LB000 ACC=LB001 DEC=LB001
' bead-perimeter_outer
MOVL C00553 V=20 PL=LB000 ACC=LB001 DEC=LB001
MOVL C00554 V=20 PL=LB000 ACC=LB001 DEC=LB001
MOVL C00555 V=20 PL=LB000 ACC=LB001 DEC=LB001
MOVL C00556 V=20 PL=LB000 ACC=LB001 DEC=LB001
' rapid-leaky
MOVL C00557 V=17 PL=LB000 ACC=LB001 DEC=LB001
' bead-solid_infill
MOVL C00558 V=20 PL=LB000 ACC=LB001 DEC=LB001
MOVL C00559 V=20 PL=LB000 ACC=LB001 DEC=LB001
MOVL C00560 V=20 PL=LB000 ACC=LB001 DEC=LB001
MOVL C00561 V=20 PL=LB000 ACC=LB001 DEC=LB001
MOVL C00562 V=20 PL=LB000 ACC=LB001 DEC=LB001
MOVL C00563 V=20 PL=LB000 ACC=LB001 DEC=LB001
MOVL C00564 V=20 PL=LB000 ACC=LB001 DEC=LB001
MOVL C00565 V=20 PL=LB000 ACC=LB001 DEC=LB001
MOVL C00566 V=20 PL=LB000 ACC=LB001 DEC=LB001
MOVL C00567 V=20 PL=LB000 ACC=LB001 DEC=LB001
MOVL C00568 V=20 PL=LB000 ACC=LB001 DEC=LB001
MOVL C00569 V=20 PL=LB000 ACC=LB001 DEC=LB001
MOVL C00570 V=20 PL=LB000 ACC=LB001 DEC=LB001
MOVL C00571 V=20 PL=LB000 ACC=LB001 DEC=LB001
MOVL C00572 V=20 PL=LB000 ACC=LB001 DEC=LB001
MOVL C00573 V=20 PL=LB000 ACC=LB001 DEC=LB001
MOVL C00574 V=20 PL=LB000 ACC=LB001 DEC=LB001
MOVL C00575 V=20 PL=LB000 ACC=LB001 DEC=LB001
MOVL C00576 V=20 PL=LB000 ACC=LB001 DEC=LB001
MOVL C00577 V=20 PL=LB000 ACC=LB001 DEC=LB001
MOVL C00578 V=20 PL=LB000 ACC=LB001 DEC=LB001
MOVL C00579 V=20 PL=LB000 ACC=LB001 DEC=LB001
MOVL C00580 V=20 PL=LB000 ACC=LB001 DEC=LB001
MOVL C00581 V=20 PL=LB000 ACC=LB001 DEC=LB001
MOVL C00582 V=20 PL=LB000 ACC=LB001 DEC=LB001
MOVL C00583 V=20 PL=LB000 ACC=LB001 DEC=LB001
MOVL C00584 V=20 PL=LB000 ACC=LB001 DEC=LB001
MOVL C00585 V=20 PL=LB000 ACC=LB001 DEC=LB001
MOVL C00586 V=20 PL=LB000 ACC=LB001 DEC=LB001
MOVL C00587 V=20 PL=LB000 ACC=LB001 DEC=LB001
MOVL C00588 V=20 PL=LB000 ACC=LB001 DEC=LB001
MOVL C00589 V=20 PL=LB000 ACC=LB001 DEC=LB001
MOVL C00590 V=25 PL=LB000 ACC=LB001 DEC=LB001
' rapid-dry
MOVL C00591 V=17 PL=LB000 ACC=LB001 DEC=LB001
MOVL C00592 V=25 PL=LB000 ACC=LB001 DEC=LB001
' bead-perimeter_outer
MOVL C00593 V=20 PL=LB000 ACC=LB001 DEC=LB001
MOVL C00594 V=20 PL=LB000 ACC=LB001 DEC=LB001
MOVL C00595 V=20 PL=LB000 ACC=LB001 DEC=LB001
MOVL C00596 V=20 PL=LB000 ACC=LB001 DEC=LB001
' rapid-leaky
MOVL C00597 V=17 PL=LB000 ACC=LB001 DEC=LB001
' bead-solid_infill
MOVL C00598 V=20 PL=LB000 ACC=LB001 DEC=LB001
MOVL C00599 V=20 PL=LB000 ACC=LB001 DEC=LB001
MOVL C00600 V=20 PL=LB000 ACC=LB001 DEC=LB001
MOVL C00601 V=20 PL=LB000 ACC=LB001 DEC=LB001
MOVL C00602 V=20 PL=LB000 ACC=LB001 DEC=LB001
MOVL C00603 V=20 PL=LB000 ACC=LB001 DEC=LB001
MOVL C00604 V=20 PL=LB000 ACC=LB001 DEC=LB001
MOVL C00605 V=20 PL=LB000 ACC=LB001 DEC=LB001
MOVL C00606 V=20 PL=LB000 ACC=LB001 DEC=LB001
MOVL C00607 V=20 PL=LB000 ACC=LB001 DEC=LB001
MOVL C00608 V=20 PL=LB000 ACC=LB001 DEC=LB001
MOVL C00609 V=20 PL=LB000 ACC=LB001 DEC=LB001
MOVL C00610 V=20 PL=LB000 ACC=LB001 DEC=LB001
MOVL C00611 V=20 PL=LB000 ACC=LB001 DEC=LB001
MOVL C00612 V=20 PL=LB000 ACC=LB001 DEC=LB001
MOVL C00613 V=20 PL=LB000 ACC=LB001 DEC=LB001
MOVL C00614 V=20 PL=LB000 ACC=LB001 DEC=LB001
MOVL C00615 V=20 PL=LB000 ACC=LB001 DEC=LB001
MOVL C00616 V=20 PL=LB000 ACC=LB001 DEC=LB001
MOVL C00617 V=20 PL=LB000 ACC=LB001 DEC=LB001
MOVL C00618 V=20 PL=LB000 ACC=LB001 DEC=LB001
MOVL C00619 V=20 PL=LB000 ACC=LB001 DEC=LB001
MOVL C00620 V=20 PL=LB000 ACC=LB001 DEC=LB001
MOVL C00621 V=20 PL=LB000 ACC=LB001 DEC=LB001
MOVL C00622 V=20 PL=LB000 ACC=LB001 DEC=LB001
MOVL C00623 V=20 PL=LB000 ACC=LB001 DEC=LB001
MOVL C00624 V=20 PL=LB000 ACC=LB001 DEC=LB001
MOVL C00625 V=20 PL=LB000 ACC=LB001 DEC=LB001
MOVL C00626 V=20 PL=LB000 ACC=LB001 DEC=LB001
MOVL C00627 V=20 PL=LB000 ACC=LB001 DEC=LB001
MOVL C00628 V=20 PL=LB000 ACC=LB001 DEC=LB001
MOVL C00629 V=20 PL=LB000 ACC=LB001 DEC=LB001
MOVL C00630 V=25 PL=LB000 ACC=LB001 DEC=LB001
' rapid-leaky
MOVL C00631 V=17 PL=LB000 ACC=LB001 DEC=LB001
MOVL C00632 V=25 PL=LB000 ACC=LB001 DEC=LB001
' bead-perimeter_outer
MOVL C00633 V=20 PL=LB000 ACC=LB001 DEC=LB001
MOVL C00634 V=20 PL=LB000 ACC=LB001 DEC=LB001
MOVL C00635 V=20 PL=LB000 ACC=LB001 DEC=LB001
MOVL C00636 V=20 PL=LB000 ACC=LB001 DEC=LB001
' rapid-leaky
MOVL C00637 V=17 PL=LB000 ACC=LB001 DEC=LB001
' bead-solid_infill
MOVL C00638 V=20 PL=LB000 ACC=LB001 DEC=LB001
MOVL C00639 V=20 PL=LB000 ACC=LB001 DEC=LB001
MOVL C00640 V=20 PL=LB000 ACC=LB001 DEC=LB001
MOVL C00641 V=20 PL=LB000 ACC=LB001 DEC=LB001
MOVL C00642 V=20 PL=LB000 ACC=LB001 DEC=LB001
MOVL C00643 V=20 PL=LB000 ACC=LB001 DEC=LB001
MOVL C00644 V=20 PL=LB000 ACC=LB001 DEC=LB001
MOVL C00645 V=20 PL=LB000 ACC=LB001 DEC=LB001
MOVL C00646 V=20 PL=LB000 ACC=LB001 DEC=LB001
MOVL C00647 V=20 PL=LB000 ACC=LB001 DEC=LB001
MOVL C00648 V=20 PL=LB000 ACC=LB001 DEC=LB001
MOVL C00649 V=20 PL=LB000 ACC=LB001 DEC=LB001
MOVL C00650 V=20 PL=LB000 ACC=LB001 DEC=LB001
MOVL C00651 V=20 PL=LB000 ACC=LB001 DEC=LB001
MOVL C00652 V=20 PL=LB000 ACC=LB001 DEC=LB001
MOVL C00653 V=20 PL=LB000 ACC=LB001 DEC=LB001
MOVL C00654 V=20 PL=LB000 ACC=LB001 DEC=LB001
MOVL C00655 V=20 PL=LB000 ACC=LB001 DEC=LB001
MOVL C00656 V=20 PL=LB000 ACC=LB001 DEC=LB001
MOVL C00657 V=20 PL=LB000 ACC=LB001 DEC=LB001
MOVL C00658 V=20 PL=LB000 ACC=LB001 DEC=LB001
MOVL C00659 V=20 PL=LB000 ACC=LB001 DEC=LB001
MOVL C00660 V=20 PL=LB000 ACC=LB001 DEC=LB001
MOVL C00661 V=20 PL=LB000 ACC=LB001 DEC=LB001
MOVL C00662 V=20 PL=LB000 ACC=LB001 DEC=LB001
MOVL C00663 V=20 PL=LB000 ACC=LB001 DEC=LB001
MOVL C00664 V=20 PL=LB000 ACC=LB001 DEC=LB001
MOVL C00665 V=20 PL=LB000 ACC=LB001 DEC=LB001
MOVL C00666 V=20 PL=LB000 ACC=LB001 DEC=LB001
MOVL C00667 V=20 PL=LB000 ACC=LB001 DEC=LB001
MOVL C00668 V=20 PL=LB000 ACC=LB001 DEC=LB001
MOVL C00669 V=20 PL=LB000 ACC=LB001 DEC=LB001
MOVL C00670 V=20 PL=LB000 ACC=LB001 DEC=LB001
MOVL C00671 V=25 PL=LB000 ACC=LB001 DEC=LB001
' rapid-leaky
MOVL C00672 V=17 PL=LB000 ACC=LB001 DEC=LB001
MOVL C00673 V=25 PL=LB000 ACC=LB001 DEC=LB001
' bead-perimeter_outer
MOVL C00674 V=20 PL=LB000 ACC=LB001 DEC=LB001
MOVL C00675 V=20 PL=LB000 ACC=LB001 DEC=LB001
MOVL C00676 V=20 PL=LB000 ACC=LB001 DEC=LB001
MOVL C00677 V=20 PL=LB000 ACC=LB001 DEC=LB001
' rapid-leaky
MOVL C00678 V=17 PL=LB000 ACC=LB001 DEC=LB001
' bead-solid_infill
MOVL C00679 V=20 PL=LB000 ACC=LB001 DEC=LB001
MOVL C00680 V=20 PL=LB000 ACC=LB001 DEC=LB001
MOVL C00681 V=20 PL=LB000 ACC=LB001 DEC=LB001
MOVL C00682 V=20 PL=LB000 ACC=LB001 DEC=LB001
MOVL C00683 V=20 PL=LB000 ACC=LB001 DEC=LB001
MOVL C00684 V=20 PL=LB000 ACC=LB001 DEC=LB001
MOVL C00685 V=20 PL=LB000 ACC=LB001 DEC=LB001
MOVL C00686 V=20 PL=LB000 ACC=LB001 DEC=LB001
MOVL C00687 V=20 PL=LB000 ACC=LB001 DEC=LB001
MOVL C00688 V=20 PL=LB000 ACC=LB001 DEC=LB001
MOVL C00689 V=20 PL=LB000 ACC=LB001 DEC=LB001
MOVL C00690 V=20 PL=LB000 ACC=LB001 DEC=LB001
MOVL C00691 V=20 PL=LB000 ACC=LB001 DEC=LB001
MOVL C00692 V=20 PL=LB000 ACC=LB001 DEC=LB001
MOVL C00693 V=20 PL=LB000 ACC=LB001 DEC=LB001
MOVL C00694 V=20 PL=LB000 ACC=LB001 DEC=LB001
MOVL C00695 V=20 PL=LB000 ACC=LB001 DEC=LB001
MOVL C00696 V=20 PL=LB000 ACC=LB001 DEC=LB001
MOVL C00697 V=20 PL=LB000 ACC=LB001 DEC=LB001
MOVL C00698 V=20 PL=LB000 ACC=LB001 DEC=LB001
MOVL C00699 V=20 PL=LB000 ACC=LB001 DEC=LB001
MOVL C00700 V=20 PL=LB000 ACC=LB001 DEC=LB001
MOVL C00701 V=20 PL=LB000 ACC=LB001 DEC=LB001
MOVL C00702 V=20 PL=LB000 ACC=LB001 DEC=LB001
MOVL C00703 V=20 PL=LB000 ACC=LB001 DEC=LB001
MOVL C00704 V=20 PL=LB000 ACC=LB001 DEC=LB001
MOVL C00705 V=20 PL=LB000 ACC=LB001 DEC=LB001
MOVL C00706 V=20 PL=LB000 ACC=LB001 DEC=LB001
MOVL C00707 V=20 PL=LB000 ACC=LB001 DEC=LB001
MOVL C00708 V=20 PL=LB000 ACC=LB001 DEC=LB001
MOVL C00709 V=20 PL=LB000 ACC=LB001 DEC=LB001
MOVL C00710 V=20 PL=LB000 ACC=LB001 DEC=LB001
MOVL C00711 V=20 PL=LB000 ACC=LB001 DEC=LB001
MOVL C00712 V=20 PL=LB000 ACC=LB001 DEC=LB001
MOVL C00713 V=20 PL=LB000 ACC=LB001 DEC=LB001
MOVL C00714 V=25 PL=LB000 ACC=LB001 DEC=LB001
' rapid-leaky
MOVL C00715 V=17 PL=LB000 ACC=LB001 DEC=LB001
MOVL C00716 V=25 PL=LB000 ACC=LB001 DEC=LB001
' bead-perimeter_outer
MOVL C00717 V=20 PL=LB000 ACC=LB001 DEC=LB001
MOVL C00718 V=20 PL=LB000 ACC=LB001 DEC=LB001
MOVL C00719 V=20 PL=LB000 ACC=LB001 DEC=LB001
MOVL C00720 V=20 PL=LB000 ACC=LB001 DEC=LB001
' rapid-leaky
MOVL C00721 V=17 PL=LB000 ACC=LB001 DEC=LB001
' bead-solid_infill
MOVL C00722 V=20 PL=LB000 ACC=LB001 DEC=LB001
MOVL C00723 V=20 PL=LB000 ACC=LB001 DEC=LB001
MOVL C00724 V=20 PL=LB000 ACC=LB001 DEC=LB001
MOVL C00725 V=20 PL=LB000 ACC=LB001 DEC=LB001
MOVL C00726 V=20 PL=LB000 ACC=LB001 DEC=LB001
MOVL C00727 V=20 PL=LB000 ACC=LB001 DEC=LB001
MOVL C00728 V=20 PL=LB000 ACC=LB001 DEC=LB001
MOVL C00729 V=20 PL=LB000 ACC=LB001 DEC=LB001
MOVL C00730 V=20 PL=LB000 ACC=LB001 DEC=LB001
MOVL C00731 V=20 PL=LB000 ACC=LB001 DEC=LB001
MOVL C00732 V=20 PL=LB000 ACC=LB001 DEC=LB001
MOVL C00733 V=20 PL=LB000 ACC=LB001 DEC=LB001
MOVL C00734 V=20 PL=LB000 ACC=LB001 DEC=LB001
MOVL C00735 V=20 PL=LB000 ACC=LB001 DEC=LB001
MOVL C00736 V=20 PL=LB000 ACC=LB001 DEC=LB001
MOVL C00737 V=20 PL=LB000 ACC=LB001 DEC=LB001
MOVL C00738 V=20 PL=LB000 ACC=LB001 DEC=LB001
MOVL C00739 V=20 PL=LB000 ACC=LB001 DEC=LB001
MOVL C00740 V=20 PL=LB000 ACC=LB001 DEC=LB001
MOVL C00741 V=20 PL=LB000 ACC=LB001 DEC=LB001
MOVL C00742 V=20 PL=LB000 ACC=LB001 DEC=LB001
MOVL C00743 V=20 PL=LB000 ACC=LB001 DEC=LB001
MOVL C00744 V=20 PL=LB000 ACC=LB001 DEC=LB001
MOVL C00745 V=20 PL=LB000 ACC=LB001 DEC=LB001
MOVL C00746 V=20 PL=LB000 ACC=LB001 DEC=LB001
MOVL C00747 V=20 PL=LB000 ACC=LB001 DEC=LB001
MOVL C00748 V=20 PL=LB000 ACC=LB001 DEC=LB001
MOVL C00749 V=20 PL=LB000 ACC=LB001 DEC=LB001
MOVL C00750 V=20 PL=LB000 ACC=LB001 DEC=LB001
MOVL C00751 V=20 PL=LB000 ACC=LB001 DEC=LB001
MOVL C00752 V=20 PL=LB000 ACC=LB001 DEC=LB001
MOVL C00753 V=25 PL=LB000 ACC=LB001 DEC=LB001
' rapid-dry
MOVL C00754 V=17 PL=LB000 ACC=LB001 DEC=LB001
MOVL C00755 V=25 PL=LB000 ACC=LB001 DEC=LB001
' bead-perimeter_outer
MOVL C00756 V=20 PL=LB000 ACC=LB001 DEC=LB001
MOVL C00757 V=20 PL=LB000 ACC=LB001 DEC=LB001
MOVL C00758 V=20 PL=LB000 ACC=LB001 DEC=LB001
MOVL C00759 V=20 PL=LB000 ACC=LB001 DEC=LB001
' rapid-leaky
MOVL C00760 V=17 PL=LB000 ACC=LB001 DEC=LB001
' bead-solid_infill
MOVL C00761 V=20 PL=LB000 ACC=LB001 DEC=LB001
MOVL C00762 V=20 PL=LB000 ACC=LB001 DEC=LB001
MOVL C00763 V=20 PL=LB000 ACC=LB001 DEC=LB001
MOVL C00764 V=20 PL=LB000 ACC=LB001 DEC=LB001
MOVL C00765 V=20 PL=LB000 ACC=LB001 DEC=LB001
MOVL C00766 V=20 PL=LB000 ACC=LB001 DEC=LB001
MOVL C00767 V=20 PL=LB000 ACC=LB001 DEC=LB001
MOVL C00768 V=20 PL=LB000 ACC=LB001 DEC=LB001
MOVL C00769 V=20 PL=LB000 ACC=LB001 DEC=LB001
MOVL C00770 V=20 PL=LB000 ACC=LB001 DEC=LB001
MOVL C00771 V=20 PL=LB000 ACC=LB001 DEC=LB001
MOVL C00772 V=20 PL=LB000 ACC=LB001 DEC=LB001
MOVL C00773 V=20 PL=LB000 ACC=LB001 DEC=LB001
MOVL C00774 V=20 PL=LB000 ACC=LB001 DEC=LB001
MOVL C00775 V=20 PL=LB000 ACC=LB001 DEC=LB001
MOVL C00776 V=20 PL=LB000 ACC=LB001 DEC=LB001
MOVL C00777 V=20 PL=LB000 ACC=LB001 DEC=LB001
MOVL C00778 V=20 PL=LB000 ACC=LB001 DEC=LB001
MOVL C00779 V=20 PL=LB000 ACC=LB001 DEC=LB001
MOVL C00780 V=20 PL=LB000 ACC=LB001 DEC=LB001
MOVL C00781 V=20 PL=LB000 ACC=LB001 DEC=LB001
MOVL C00782 V=20 PL=LB000 ACC=LB001 DEC=LB001
MOVL C00783 V=20 PL=LB000 ACC=LB001 DEC=LB001
MOVL C00784 V=20 PL=LB000 ACC=LB001 DEC=LB001
MOVL C00785 V=20 PL=LB000 ACC=LB001 DEC=LB001
MOVL C00786 V=20 PL=LB000 ACC=LB001 DEC=LB001
MOVL C00787 V=20 PL=LB000 ACC=LB001 DEC=LB001
MOVL C00788 V=20 PL=LB000 ACC=LB001 DEC=LB001
MOVL C00789 V=20 PL=LB000 ACC=LB001 DEC=LB001
MOVL C00790 V=20 PL=LB000 ACC=LB001 DEC=LB001
MOVL C00791 V=20 PL=LB000 ACC=LB001 DEC=LB001
MOVL C00792 V=25 PL=LB000 ACC=LB001 DEC=LB001
' rapid-leaky
MOVL C00793 V=17 PL=LB000 ACC=LB001 DEC=LB001
MOVL C00794 V=25 PL=LB000 ACC=LB001 DEC=LB001
' bead-perimeter_outer
MOVL C00795 V=20 PL=LB000 ACC=LB001 DEC=LB001
MOVL C00796 V=20 PL=LB000 ACC=LB001 DEC=LB001
MOVL C00797 V=20 PL=LB000 ACC=LB001 DEC=LB001
MOVL C00798 V=20 PL=LB000 ACC=LB001 DEC=LB001
MOVL C00799 V=25 PL=LB000 ACC=LB001 DEC=LB001
' rapid-dry
MOVL C00800 V=17 PL=LB000 ACC=LB001 DEC=LB001
MOVL C00801 V=25 PL=LB000 ACC=LB001 DEC=LB001
' bead-solid_infill
MOVL C00802 V=20 PL=LB000 ACC=LB001 DEC=LB001
MOVL C00803 V=20 PL=LB000 ACC=LB001 DEC=LB001
MOVL C00804 V=20 PL=LB000 ACC=LB001 DEC=LB001
MOVL C00805 V=20 PL=LB000 ACC=LB001 DEC=LB001
MOVL C00806 V=20 PL=LB000 ACC=LB001 DEC=LB001
MOVL C00807 V=20 PL=LB000 ACC=LB001 DEC=LB001
MOVL C00808 V=20 PL=LB000 ACC=LB001 DEC=LB001
MOVL C00809 V=20 PL=LB000 ACC=LB001 DEC=LB001
MOVL C00810 V=20 PL=LB000 ACC=LB001 DEC=LB001
MOVL C00811 V=20 PL=LB000 ACC=LB001 DEC=LB001
MOVL C00812 V=20 PL=LB000 ACC=LB001 DEC=LB001
MOVL C00813 V=20 PL=LB000 ACC=LB001 DEC=LB001
MOVL C00814 V=20 PL=LB000 ACC=LB001 DEC=LB001
MOVL C00815 V=20 PL=LB000 ACC=LB001 DEC=LB001
MOVL C00816 V=20 PL=LB000 ACC=LB001 DEC=LB001
MOVL C00817 V=20 PL=LB000 ACC=LB001 DEC=LB001
MOVL C00818 V=20 PL=LB000 ACC=LB001 DEC=LB001
MOVL C00819 V=20 PL=LB000 ACC=LB001 DEC=LB001
MOVL C00820 V=20 PL=LB000 ACC=LB001 DEC=LB001
MOVL C00821 V=20 PL=LB000 ACC=LB001 DEC=LB001
MOVL C00822 V=20 PL=LB000 ACC=LB001 DEC=LB001
MOVL C00823 V=20 PL=LB000 ACC=LB001 DEC=LB001
MOVL C00824 V=20 PL=LB000 ACC=LB001 DEC=LB001
MOVL C00825 V=20 PL=LB000 ACC=LB001 DEC=LB001
MOVL C00826 V=20 PL=LB000 ACC=LB001 DEC=LB001
MOVL C00827 V=20 PL=LB000 ACC=LB001 DEC=LB001
MOVL C00828 V=20 PL=LB000 ACC=LB001 DEC=LB001
MOVL C00829 V=20 PL=LB000 ACC=LB001 DEC=LB001
MOVL C00830 V=20 PL=LB000 ACC=LB001 DEC=LB001
MOVL C00831 V=20 PL=LB000 ACC=LB001 DEC=LB001
MOVL C00832 V=20 PL=LB000 ACC=LB001 DEC=LB001
MOVL C00833 V=20 PL=LB000 ACC=LB001 DEC=LB001
MOVL C00834 V=25 PL=LB000 ACC=LB001 DEC=LB001
' rapid-leaky
MOVL C00835 V=17 PL=LB000 ACC=LB001 DEC=LB001
MOVL C00836 V=25 PL=LB000 ACC=LB001 DEC=LB001
' bead-perimeter_outer
MOVL C00837 V=20 PL=LB000 ACC=LB001 DEC=LB001
MOVL C00838 V=20 PL=LB000 ACC=LB001 DEC=LB001
MOVL C00839 V=20 PL=LB000 ACC=LB001 DEC=LB001
MOVL C00840 V=20 PL=LB000 ACC=LB001 DEC=LB001
' rapid-leaky
MOVL C00841 V=17 PL=LB000 ACC=LB001 DEC=LB001
' bead-solid_infill
MOVL C00842 V=20 PL=LB000 ACC=LB001 DEC=LB001
MOVL C00843 V=20 PL=LB000 ACC=LB001 DEC=LB001
MOVL C00844 V=20 PL=LB000 ACC=LB001 DEC=LB001
MOVL C00845 V=20 PL=LB000 ACC=LB001 DEC=LB001
MOVL C00846 V=20 PL=LB000 ACC=LB001 DEC=LB001
MOVL C00847 V=20 PL=LB000 ACC=LB001 DEC=LB001
MOVL C00848 V=20 PL=LB000 ACC=LB001 DEC=LB001
MOVL C00849 V=20 PL=LB000 ACC=LB001 DEC=LB001
MOVL C00850 V=20 PL=LB000 ACC=LB001 DEC=LB001
MOVL C00851 V=20 PL=LB000 ACC=LB001 DEC=LB001
MOVL C00852 V=20 PL=LB000 ACC=LB001 DEC=LB001
MOVL C00853 V=20 PL=LB000 ACC=LB001 DEC=LB001
MOVL C00854 V=20 PL=LB000 ACC=LB001 DEC=LB001
MOVL C00855 V=20 PL=LB000 ACC=LB001 DEC=LB001
MOVL C00856 V=20 PL=LB000 ACC=LB001 DEC=LB001
MOVL C00857 V=20 PL=LB000 ACC=LB001 DEC=LB001
MOVL C00858 V=20 PL=LB000 ACC=LB001 DEC=LB001
MOVL C00859 V=20 PL=LB000 ACC=LB001 DEC=LB001
MOVL C00860 V=20 PL=LB000 ACC=LB001 DEC=LB001
MOVL C00861 V=20 PL=LB000 ACC=LB001 DEC=LB001
MOVL C00862 V=20 PL=LB000 ACC=LB001 DEC=LB001
MOVL C00863 V=20 PL=LB000 ACC=LB001 DEC=LB001
MOVL C00864 V=20 PL=LB000 ACC=LB001 DEC=LB001
MOVL C00865 V=20 PL=LB000 ACC=LB001 DEC=LB001
MOVL C00866 V=20 PL=LB000 ACC=LB001 DEC=LB001
MOVL C00867 V=20 PL=LB000 ACC=LB001 DEC=LB001
MOVL C00868 V=20 PL=LB000 ACC=LB001 DEC=LB001
MOVL C00869 V=20 PL=LB000 ACC=LB001 DEC=LB001
MOVL C00870 V=20 PL=LB000 ACC=LB001 DEC=LB001
MOVL C00871 V=20 PL=LB000 ACC=LB001 DEC=LB001
MOVL C00872 V=20 PL=LB000 ACC=LB001 DEC=LB001
MOVL C00873 V=20 PL=LB000 ACC=LB001 DEC=LB001
MOVL C00874 V=25 PL=LB000 ACC=LB001 DEC=LB001
' rapid-leaky
MOVL C00875 V=17 PL=LB000 ACC=LB001 DEC=LB001
MOVL C00876 V=25 PL=LB000 ACC=LB001 DEC=LB001
' bead-perimeter_outer
MOVL C00877 V=20 PL=LB000 ACC=LB001 DEC=LB001
MOVL C00878 V=20 PL=LB000 ACC=LB001 DEC=LB001
MOVL C00879 V=20 PL=LB000 ACC=LB001 DEC=LB001
MOVL C00880 V=20 PL=LB000 ACC=LB001 DEC=LB001
' rapid-leaky
MOVL C00881 V=17 PL=LB000 ACC=LB001 DEC=LB001
' bead-solid_infill
MOVL C00882 V=20 PL=LB000 ACC=LB001 DEC=LB001
MOVL C00883 V=20 PL=LB000 ACC=LB001 DEC=LB001
MOVL C00884 V=20 PL=LB000 ACC=LB001 DEC=LB001
MOVL C00885 V=20 PL=LB000 ACC=LB001 DEC=LB001
MOVL C00886 V=20 PL=LB000 ACC=LB001 DEC=LB001
MOVL C00887 V=20 PL=LB000 ACC=LB001 DEC=LB001
MOVL C00888 V=20 PL=LB000 ACC=LB001 DEC=LB001
MOVL C00889 V=20 PL=LB000 ACC=LB001 DEC=LB001
MOVL C00890 V=20 PL=LB000 ACC=LB001 DEC=LB001
MOVL C00891 V=20 PL=LB000 ACC=LB001 DEC=LB001
MOVL C00892 V=20 PL=LB000 ACC=LB001 DEC=LB001
MOVL C00893 V=20 PL=LB000 ACC=LB001 DEC=LB001
MOVL C00894 V=20 PL=LB000 ACC=LB001 DEC=LB001
MOVL C00895 V=20 PL=LB000 ACC=LB001 DEC=LB001
MOVL C00896 V=20 PL=LB000 ACC=LB001 DEC=LB001
MOVL C00897 V=20 PL=LB000 ACC=LB001 DEC=LB001
MOVL C00898 V=20 PL=LB000 ACC=LB001 DEC=LB001
MOVL C00899 V=20 PL=LB000 ACC=LB001 DEC=LB001
MOVL C00900 V=20 PL=LB000 ACC=LB001 DEC=LB001
MOVL C00901 V=20 PL=LB000 ACC=LB001 DEC=LB001
MOVL C00902 V=20 PL=LB000 ACC=LB001 DEC=LB001
MOVL C00903 V=20 PL=LB000 ACC=LB001 DEC=LB001
MOVL C00904 V=20 PL=LB000 ACC=LB001 DEC=LB001
MOVL C00905 V=20 PL=LB000 ACC=LB001 DEC=LB001
MOVL C00906 V=20 PL=LB000 ACC=LB001 DEC=LB001
MOVL C00907 V=20 PL=LB000 ACC=LB001 DEC=LB001
MOVL C00908 V=20 PL=LB000 ACC=LB001 DEC=LB001
MOVL C00909 V=20 PL=LB000 ACC=LB001 DEC=LB001
MOVL C00910 V=20 PL=LB000 ACC=LB001 DEC=LB001
MOVL C00911 V=20 PL=LB000 ACC=LB001 DEC=LB001
MOVL C00912 V=20 PL=LB000 ACC=LB001 DEC=LB001
MOVL C00913 V=20 PL=LB000 ACC=LB001 DEC=LB001
MOVL C00914 V=20 PL=LB000 ACC=LB001 DEC=LB001
MOVL C00915 V=25 PL=LB000 ACC=LB001 DEC=LB001
' rapid-dry
MOVL C00916 V=17 PL=LB000 ACC=LB001 DEC=LB001
MOVL C00917 V=25 PL=LB000 ACC=LB001 DEC=LB001
' bead-perimeter_outer
MOVL C00918 V=20 PL=LB000 ACC=LB001 DEC=LB001
MOVL C00919 V=20 PL=LB000 ACC=LB001 DEC=LB001
MOVL C00920 V=20 PL=LB000 ACC=LB001 DEC=LB001
MOVL C00921 V=20 PL=LB000 ACC=LB001 DEC=LB001
' rapid-leaky
MOVL C00922 V=17 PL=LB000 ACC=LB001 DEC=LB001
' bead-solid_infill
MOVL C00923 V=20 PL=LB000 ACC=LB001 DEC=LB001
MOVL C00924 V=20 PL=LB000 ACC=LB001 DEC=LB001
MOVL C00925 V=20 PL=LB000 ACC=LB001 DEC=LB001
MOVL C00926 V=20 PL=LB000 ACC=LB001 DEC=LB001
MOVL C00927 V=20 PL=LB000 ACC=LB001 DEC=LB001
MOVL C00928 V=20 PL=LB000 ACC=LB001 DEC=LB001
MOVL C00929 V=20 PL=LB000 ACC=LB001 DEC=LB001
MOVL C00930 V=20 PL=LB000 ACC=LB001 DEC=LB001
MOVL C00931 V=20 PL=LB000 ACC=LB001 DEC=LB001
MOVL C00932 V=20 PL=LB000 ACC=LB001 DEC=LB001
MOVL C00933 V=20 PL=LB000 ACC=LB001 DEC=LB001
MOVL C00934 V=20 PL=LB000 ACC=LB001 DEC=LB001
MOVL C00935 V=20 PL=LB000 ACC=LB001 DEC=LB001
MOVL C00936 V=20 PL=LB000 ACC=LB001 DEC=LB001
MOVL C00937 V=20 PL=LB000 ACC=LB001 DEC=LB001
MOVL C00938 V=20 PL=LB000 ACC=LB001 DEC=LB001
MOVL C00939 V=20 PL=LB000 ACC=LB001 DEC=LB001
MOVL C00940 V=20 PL=LB000 ACC=LB001 DEC=LB001
MOVL C00941 V=20 PL=LB000 ACC=LB001 DEC=LB001
MOVL C00942 V=20 PL=LB000 ACC=LB001 DEC=LB001
MOVL C00943 V=20 PL=LB000 ACC=LB001 DEC=LB001
MOVL C00944 V=20 PL=LB000 ACC=LB001 DEC=LB001
MOVL C00945 V=20 PL=LB000 ACC=LB001 DEC=LB001
MOVL C00946 V=20 PL=LB000 ACC=LB001 DEC=LB001
MOVL C00947 V=20 PL=LB000 ACC=LB001 DEC=LB001
MOVL C00948 V=20 PL=LB000 ACC=LB001 DEC=LB001
MOVL C00949 V=20 PL=LB000 ACC=LB001 DEC=LB001
MOVL C00950 V=20 PL=LB000 ACC=LB001 DEC=LB001
MOVL C00951 V=20 PL=LB000 ACC=LB001 DEC=LB001
MOVL C00952 V=20 PL=LB000 ACC=LB001 DEC=LB001
MOVL C00953 V=20 PL=LB000 ACC=LB001 DEC=LB001
MOVL C00954 V=20 PL=LB000 ACC=LB001 DEC=LB001
MOVL C00955 V=20 PL=LB000 ACC=LB001 DEC=LB001
MOVL C00956 V=20 PL=LB000 ACC=LB001 DEC=LB001
MOVL C00957 V=20 PL=LB000 ACC=LB001 DEC=LB001
MOVL C00958 V=25 PL=LB000 ACC=LB001 DEC=LB001
' rapid-leaky
MOVL C00959 V=17 PL=LB000 ACC=LB001 DEC=LB001
MOVL C00960 V=25 PL=LB000 ACC=LB001 DEC=LB001
' bead-perimeter_outer
MOVL C00961 V=20 PL=LB000 ACC=LB001 DEC=LB001
MOVL C00962 V=20 PL=LB000 ACC=LB001 DEC=LB001
MOVL C00963 V=20 PL=LB000 ACC=LB001 DEC=LB001
MOVL C00964 V=20 PL=LB000 ACC=LB001 DEC=LB001
' rapid-leaky
MOVL C00965 V=17 PL=LB000 ACC=LB001 DEC=LB001
' bead-solid_infill
MOVL C00966 V=20 PL=LB000 ACC=LB001 DEC=LB001
MOVL C00967 V=20 PL=LB000 ACC=LB001 DEC=LB001
MOVL C00968 V=20 PL=LB000 ACC=LB001 DEC=LB001
MOVL C00969 V=20 PL=LB000 ACC=LB001 DEC=LB001
MOVL C00970 V=20 PL=LB000 ACC=LB001 DEC=LB001
MOVL C00971 V=20 PL=LB000 ACC=LB001 DEC=LB001
MOVL C00972 V=20 PL=LB000 ACC=LB001 DEC=LB001
MOVL C00973 V=20 PL=LB000 ACC=LB001 DEC=LB001
MOVL C00974 V=20 PL=LB000 ACC=LB001 DEC=LB001
MOVL C00975 V=20 PL=LB000 ACC=LB001 DEC=LB001
MOVL C00976 V=20 PL=LB000 ACC=LB001 DEC=LB001
MOVL C00977 V=20 PL=LB000 ACC=LB001 DEC=LB001
MOVL C00978 V=20 PL=LB000 ACC=LB001 DEC=LB001
MOVL C00979 V=20 PL=LB000 ACC=LB001 DEC=LB001
MOVL C00980 V=20 PL=LB000 ACC=LB001 DEC=LB001
MOVL C00981 V=20 PL=LB000 ACC=LB001 DEC=LB001
MOVL C00982 V=20 PL=LB000 ACC=LB001 DEC=LB001
MOVL C00983 V=20 PL=LB000 ACC=LB001 DEC=LB001
MOVL C00984 V=20 PL=LB000 ACC=LB001 DEC=LB001
MOVL C00985 V=20 PL=LB000 ACC=LB001 DEC=LB001
MOVL C00986 V=20 PL=LB000 ACC=LB001 DEC=LB001
MOVL C00987 V=20 PL=LB000 ACC=LB001 DEC=LB001
MOVL C00988 V=20 PL=LB000 ACC=LB001 DEC=LB001
MOVL C00989 V=20 PL=LB000 ACC=LB001 DEC=LB001
MOVL C00990 V=20 PL=LB000 ACC=LB001 DEC=LB001
MOVL C00991 V=20 PL=LB000 ACC=LB001 DEC=LB001
MOVL C00992 V=20 PL=LB000 ACC=LB001 DEC=LB001
MOVL C00993 V=20 PL=LB000 ACC=LB001 DEC=LB001
MOVL C00994 V=20 PL=LB000 ACC=LB001 DEC=LB001
MOVL C00995 V=20 PL=LB000 ACC=LB001 DEC=LB001
MOVL C00996 V=20 PL=LB000 ACC=LB001 DEC=LB001
MOVL C00997 V=25 PL=LB000 ACC=LB001 DEC=LB001
' rapid-leaky
MOVL C00998 V=17 PL=LB000 ACC=LB001 DEC=LB001
MOVL C00999 V=25 PL=LB000 ACC=LB001 DEC=LB001
' bead-perimeter_outer
MOVL C01000 V=20 PL=LB000 ACC=LB001 DEC=LB001
MOVL C01001 V=20 PL=LB000 ACC=LB001 DEC=LB001
MOVL C01002 V=20 PL=LB000 ACC=LB001 DEC=LB001
MOVL C01003 V=20 PL=LB000 ACC=LB001 DEC=LB001
' rapid-leaky
MOVL C01004 V=17 PL=LB000 ACC=LB001 DEC=LB001
' bead-sparse_infill
MOVL C01005 V=20 PL=LB000 ACC=LB001 DEC=LB001
MOVL C01006 V=20 PL=LB000 ACC=LB001 DEC=LB001
MOVL C01007 V=20 PL=LB000 ACC=LB001 DEC=LB001
MOVL C01008 V=20 PL=LB000 ACC=LB001 DEC=LB001
MOVL C01009 V=20 PL=LB000 ACC=LB001 DEC=LB001
MOVL C01010 V=20 PL=LB000 ACC=LB001 DEC=LB001
